// TwinCAT 3 PLC project StageCore
// Title: StageCore
// Company: _
// Author: Krystian Lis et al.
// ProjectVersion: 6.0.0
// ProgramVersion: 3.1.4026.18
// libraries:
//   Tc2_Math, * (Beckhoff Automation GmbH)
//   Tc2_Standard, * (Beckhoff Automation GmbH)
//   Tc2_System, * (Beckhoff Automation GmbH)
//   Tc2_Utilities, * (Beckhoff Automation GmbH)
// project tree:
//   Broadcast/Arg/Args/BOOL/ BoolArg.TcPOU (not stored), IArgToIBoolArg.TcPOU (not stored), I_BoolArg.TcIO (not stored)
//   Broadcast/Arg/Args/DWORD/ DwordArg.TcPOU (not stored), IArgToIDwordArg.TcPOU (not stored), I_DwordArg.TcIO (not stored)
//   Broadcast/Arg/Args/REAL/ IArgToIRealtArg.TcPOU (not stored), I_RealArg.TcIO (not stored), RealArg.TcPOU (not stored)
//   Broadcast/Arg/ IArgToIComp.TcPOU, ICompToIArg.TcPOU (not stored), I_Arg.TcIO (not stored)
//   Broadcast/Callable/ I_Callable.TcIO (not stored)
//   Broadcast/Helpers/ GetSignal.TcPOU (not stored), GetReceiver.TcPOU
//   Broadcast/Receiver/ ICompToIRec.TcPOU (not stored), I_Receiver.TcIO, I_ReceiverNode.TcIO (not stored), Receiver.TcPOU
//   Broadcast/Signal/ ICompToISignal.TcPOU, I_SignalEmit.TcIO, I_Signal.TcIO, I_SignalNode.TcIO (not stored), Signal.TcPOU
//   Broadcast/Sys/Helpers/ _BroadcastDefragment.TcPOU, _BroadcastGetBestFit.TcPOU (not stored), _Emit.TcPOU (not stored), _Pair.TcPOU, _RegSignal.TcPOU (not stored), _Unpair.TcPOU (not stored)
//   Broadcast/Sys/Structs/ _BroadcastStruct.TcDUT (not stored), _BroadcastUnion.TcDUT (not stored)
//   Broadcast/Sys/ _Broadcast.TcGVL (not stored)
//   Dbg/ DebugInfo.TcPOU, NewDebug.TcPOU, DebugMode.TcDUT, I_Debug.TcIO (not stored), _DebugInfo.TcDUT, _Debug.TcGVL
//   Entity/Core/ Component.TcPOU, I_Component.TcIO (not stored), GetOwnerFromRaw.TcPOU, I_RawComponent.TcIO (not stored), I_Entity.TcIO, GetNextEntity.TcPOU, GetPrevEntity.TcPOU
//   Entity/Core/Scope/ EntityEnd.TcPOU, EntityExtend.TcPOU, EntityStart.TcPOU
//   Entity/Sys/ _EntityState.TcDUT (not stored), _Ec.TcGVL
//   Entity/Sys/_Helpers/ _EntityEnd.TcPOU, _EntityExtend.TcPOU (not stored), _EntityStart.TcPOU (not stored), _RegisterComponent.TcPOU
//   Entity/Sys/_Itf/ I_ComponentNode.TcIO, I_EntityNode.TcIO
//   Result/Error/ Err.TcGVL (not stored), GenericResult.TcGVL (not stored)
//   Result/ IsErr.TcPOU (not stored), IsNone.TcPOU (not stored), IsOk.TcPOU, IsFail.TcPOU, IsSome.TcPOU (not stored), IsEnd.TcPOU, Result.TcDUT (not stored), ResultToStr.TcPOU
//   Runtime/Execute/ Execute.TcPOU, I_Execute.TcIO, I_ExecuteNode.TcIO (not stored)
//   Runtime/Init/ Init.TcPOU, I_InitNode.TcIO (not stored), I_Init.TcIO (not stored)
//   Runtime/ Runtime.TcPOU, _Runtime.TcGVL (not stored)
//   State/_Buffer/ _StateBuffer.TcPOU
//   State/Helpers/ GetStateManager.TcPOU, GetState.TcPOU (not stored)
//   State/_Machine/ _StateMachine.TcPOU
//   State/Manager/ ICompToIStateMgr.TcPOU, I_StateManager.TcIO (not stored), StateManager.TcPOU
//   State/State/ ICompToIState.TcPOU (not stored), I_State.TcIO, I_StateInternal.TcIO, State.TcPOU
//   Strings/Alias/ Ch.TcDUT (not stored), Str.TcDUT (not stored)
//   Strings/Strb/ I_Strb.TcIO (not stored), Strb.TcPOU
//   Strings/Strf/ Strf.TcPOU
//   Tags/Casts/ IArgToITag.TcPOU, ICompToITag.TcPOU (not stored)
//   Tags/Helpers/ GetTag.TcPOU, GetTagOption.TcPOU, HasTagOption.TcPOU, HasTag.TcPOU (not stored), MatchPath.TcPOU
//   Tags/ I_Tag.TcIO, I_TagCmp.TcIO, TagBase.TcPOU, TagCmp.TcPOU (not stored), TagPath.TcPOU (not stored), Tag.TcPOU (not stored)
//   Jobs/Worker/Base/ Worker.TcPOU, I_Worker.TcIO
//   Jobs/Worker/ LoopWorker.TcPOU, BlockingWorker.TcPOU
//   Jobs/Job/ I_Job.TcIO, I_JobInternal.TcIO, Job.TcPOU
//   Jobs/ JobState.TcDUT
//   _/ Param.TcGVL
// (motion and I/O tree: see PLC project stageutils)
// real-time tasks:
//   TASK Example: cycle T#10ms, priority 20, ADS port 350
//   TASK Test: cycle T#10ms, priority 21, ADS port 351
//   TASK VISU_TASK: cycle T#200000us, priority 30, ADS port 352

// ---- Dbg/DebugMode.TcDUT
{attribute 'qualified_only'}
{attribute 'strict'}
{attribute 'to_string'}
TYPE DebugMode :
(
	Notify,
	Panic
) BYTE;
END_TYPE

// ---- Dbg/_DebugInfo.TcDUT
TYPE INTERNAL _DebugInfo :
STRUCT
	iDebugMain: I_Debug;
	iDebugSub: I_Debug;
	mode: DebugMode;
	sComment: Str;
END_STRUCT
END_TYPE

// ---- Jobs/JobState.TcDUT
(*
State of a Job.
*)
{attribute 'qualified_only'}
{attribute 'strict'}
TYPE JobState :
(
	Error,
	Idle,
	Enqueue,
	Ready,
	Running,
	Aborted,
	Completed
) BYTE := Idle;
END_TYPE

// ---- Dbg/_Debug.TcGVL
{attribute 'qualified_only'}
VAR_GLOBAL INTERNAL
	debugMsg: ARRAY[1..Param.DEBUG_CAP] OF _DebugInfo;	
	nLastIdx: UDINT;
	
	nTotalNumber: UDINT;
	nNotifyNumber: UDINT;
	nPanicNumber: UDINT;
END_VAR

// ---- Entity/Sys/_Ec.TcGVL
// ---------------------------------------------------------------------------
// GLOBAL DATA BLOCK: _Ec
// Purpose: Stores and manages the state and structure of all registered entities 
//          and tracks the current scope under construction.

// This attribute ensures variables are accessed using qualified names (e.g., _Ec.iFirst)
{attribute 'qualified_only'}

VAR_GLOBAL INTERNAL    
    // Reference to the first registered entity in the global entity list
    iFirst: I_Entity;

    // Reference to the last registered entity in the global entity list
    iLast: I_Entity;

    // Points to the entity currently being constructed
    // Used to add components or nested entities during initialization
    iUnderConstruction: I_Entity;

    // Tracks how many nested entity scopes are currently under construction
    // Used to manage hierarchical or recursive construction logic
    nConstructedScopes: UDINT;
END_VAR

// ---- _/Param.TcGVL
{attribute 'qualified_only'}
// DO NOT SET ANY OF THE CAP PARAMETERS TO 0 OR LARGER THAN MAX DINT!!!
VAR_GLOBAL CONSTANT
	SIGNAL_CAP		: UDINT(1..16#7FFFFFFF) := 20; // Max number of signals.
	RECEIVER_CAP	: UDINT(1..16#7FFFFFFF) := 100; // Max number of signal-receiver pairings.
	
	
	DEBUG_CAP	: UDINT(1..16#7FFFFFFF) := 10; // Max number of debug messages.
	INIT_INTERNAL_DEBUG_MODE: DebugMode := DebugMode.Panic; // Should internal debug messages during initialization stop Runtime?
	EXE_INTERNAL_DEBUG_MODE: DebugMode := DebugMode.Notify; // Should internal debug messages during execution stop Runtime?
END_VAR

// ---- Broadcast/Receiver/I_Receiver.TcIO
(*
Represents a receiver in the Broadcast system. Implements the necessary methods for receiving events and pairing signals.
Can be casted to `I_Component`.
*)
INTERFACE I_Receiver EXTENDS I_ReceiverNode, I_RawComponent

PROPERTY Tag : I_Tag
GET
END_GET
END_PROPERTY

END_INTERFACE

// ---- Broadcast/Signal/I_SignalEmit.TcIO
(*
Enables pairing with receivers and emitting, but not casting to `I_Component`.
*)
INTERFACE I_SignalEmit

(*
Emits an argument through the signal's broadcasting system.  
If no argument is provided, it defaults to emitting the associated tag.
Returns:
- `Ok` - On Success
- `Err.InfLoop` - Upon recursive call attempt
*)
METHOD Emit : Result
VAR_INPUT
	iArg			: I_Arg := 0;
END_VAR
END_METHOD

(*
Emits an argument to a specified receiver.
Returns:
- `Ok` - If the emission is successful.
- `Err.Itf0` - If the receiver interface is invalid.
- `Err.InfLoop` - Upon recursive call attempt
*)
METHOD EmitTo : Result
VAR_INPUT
	iReceiver		: I_Receiver;
	iArg			: I_Arg := 0;
END_VAR
END_METHOD

(*
Allows access to Option property of the internal Tag.
*)
PROPERTY Option : Str
GET
END_GET
SET
END_SET
END_PROPERTY

(*
Pairs the signal with a receiver.  
Returns:
- `Ok` - If pairing is successful.
- `Err.Itf0` - If the receiver interface is invalid.
- `Err.IncArg` - If the `I_Receiver` is invalid.
- `Err.ItfEq` - If the `I_Receiver` is already paired with this `I_Signal`.
- `Err.Ovf` - If there is no space for another pairing.
*)
METHOD Pair : Result
VAR_INPUT
	iReceiver		: I_Receiver;
END_VAR
END_METHOD

(*
Provides access to the tag associated with the signal.
*)
PROPERTY Tag : I_Tag
GET
END_GET
END_PROPERTY

(*
Unpairs the signal from a specified receiver.
Returns:
- `Ok` - If unpairing is successful.
- `Err.Itf0` - If the receiver interface is invalid.
- `Err.IncArg` - If the `I_Receiver` is invalid.
- `Err.NoMatch` - If `I_Signal` is not paired with this `I_Receiver`.
*)
METHOD Unpair : Result
VAR_INPUT
	iReceiver		: I_Receiver;
END_VAR
END_METHOD

END_INTERFACE

// ---- Broadcast/Signal/I_Signal.TcIO
(*
Enables pairing with receivers and casting to `I_Component`, but no emitting.
*)
INTERFACE I_Signal EXTENDS I_Debug, I_RawComponent

(*
Pairs the signal with a receiver.  
Returns:
- `Ok` - If pairing is successful.
- `Err.Itf0` - If the receiver interface is invalid.
- `Err.IncArg` - If the `I_Receiver` is invalid.
- `Err.ItfEq` - If the `I_Receiver` is already paired with this `I_Signal`.
- `Err.Ovf` - If there is no space for another pairing.
*)
METHOD Pair : Result
VAR_INPUT
	iReceiver		: I_Receiver;
END_VAR
END_METHOD

PROPERTY Tag : I_Tag
GET
END_GET
END_PROPERTY

(*
Unpairs the signal from a specified receiver.
Returns:
- `Ok` - If unpairing is successful.
- `Err.Itf0` - If the receiver interface is invalid.
- `Err.IncArg` - If the `I_Receiver` is invalid.
- `Err.NoMatch` - If `I_Signal` is not paired with this `I_Receiver`.
*)
METHOD Unpair : Result
VAR_INPUT
	iReceiver		: I_Receiver;
END_VAR
END_METHOD

END_INTERFACE

// ---- Entity/Core/I_Entity.TcIO
(*
Represents a registered entity in the Entity-Component system.
*)
INTERFACE I_Entity EXTENDS I_EntityNode

END_INTERFACE

// ---- Entity/Sys/_Itf/I_ComponentNode.TcIO
INTERFACE INTERNAL I_ComponentNode EXTENDS I_Debug

PROPERTY INTERNAL _Entity : I_Entity
GET
END_GET
SET
END_SET
END_PROPERTY

PROPERTY INTERNAL _Next : I_Component
GET
END_GET
SET
END_SET
END_PROPERTY

PROPERTY INTERNAL _Prev : I_Component
GET
END_GET
SET
END_SET
END_PROPERTY

END_INTERFACE

// ---- Entity/Sys/_Itf/I_EntityNode.TcIO
INTERFACE INTERNAL I_EntityNode EXTENDS I_Debug

PROPERTY INTERNAL _FirstComp : I_Component
GET
END_GET
SET
END_SET
END_PROPERTY

PROPERTY INTERNAL _LastComp : I_Component
GET
END_GET
SET
END_SET
END_PROPERTY

PROPERTY INTERNAL _Next : I_Entity
GET
END_GET
SET
END_SET
END_PROPERTY

PROPERTY INTERNAL _Prev : I_Entity
GET
END_GET
SET
END_SET
END_PROPERTY

PROPERTY INTERNAL _Size : UDINT
GET
END_GET
SET
END_SET
END_PROPERTY

PROPERTY INTERNAL _State : _EntityState
GET
END_GET
SET
END_SET
END_PROPERTY

(*
Description: Retrieves a previous component before the inputted one or last component if referenced value is 0.
Returns:
- Ok - Returns upon success, updates referenced value with new component.
- Err.InvRef - Invalid output reference.
- Err.ItfEq - Provided interface pointer doesn't belong to the queried entity. Nulls reference.
- Err.NotFound - The entity doesn't contain any components. Nulls reference.
- Err.End - No more components. Nulls reference.
*)
METHOD GetNextComp : Result
VAR_INPUT
	iOut		: REFERENCE TO I_Component;
END_VAR
END_METHOD

(*
Description: Retrieves a previous component before the inputted one or last component if referenced value is 0.
Returns:
- Ok - Returns upon success, updates referenced value with new component.
- Err.InvRef - Invalid output reference.
- Err.ItfEq - Provided interface pointer doesn't belong to the queried entity. Nulls reference.
- Err.NotFound - The entity doesn't contain any components. Nulls reference.
- Err.End - No more components. Nulls reference.
*)
METHOD GetPrevComp : Result
VAR_INPUT
	iOut		: REFERENCE TO I_Component;
END_VAR
END_METHOD

(*
Provides the size of the entity, indicating the number of components it manages.  
Note: For internal logic purposes, this value is incremented by one beyond the actual component count.
*)
PROPERTY Size : UDINT
GET
END_GET
END_PROPERTY

END_INTERFACE

// ---- Runtime/Execute/I_Execute.TcIO
(*
A `Execute` method of FB implmenting this interface will be called every control loop cycle.
*)
INTERFACE I_Execute EXTENDS I_Debug

(*
If registered, this method will be executed cyclically.
*)
METHOD Execute
VAR_INPUT
	nPhase: INT;
END_VAR
END_METHOD

END_INTERFACE

// ---- State/State/I_State.TcIO
(*
Allows states to be cast to `I_RawComponent`.
*)
INTERFACE I_State EXTENDS I_RawComponent, I_Debug, I_StateInternal

(*
Returns the entity that owns this state.
*)
PROPERTY Owner : I_Entity
GET
END_GET
END_PROPERTY

PROPERTY Tag : I_Tag
GET
END_GET
END_PROPERTY

END_INTERFACE

// ---- State/State/I_StateInternal.TcIO
INTERFACE INTERNAL I_StateInternal

METHOD INTERNAL _CanActivate : BOOL
VAR_INPUT
END_VAR
END_METHOD

METHOD INTERNAL _CanDeactivate : BOOL
VAR_INPUT
END_VAR
END_METHOD

PROPERTY INTERNAL _InQueue : BOOL
GET
END_GET
SET
END_SET
END_PROPERTY

PROPERTY INTERNAL _NextInBuffer : I_State
GET
END_GET
SET
END_SET
END_PROPERTY

METHOD INTERNAL _OnEntry
VAR_INPUT
END_VAR
END_METHOD

METHOD INTERNAL _OnExecute
VAR_INPUT
END_VAR
END_METHOD

METHOD INTERNAL _OnExit
VAR_INPUT
END_VAR
END_METHOD

(*
Returns the entity that owns this state.
*)
PROPERTY Owner : I_Entity
GET
END_GET
END_PROPERTY

END_INTERFACE

// ---- Tags/I_Tag.TcIO
(*
An identifier that uses reflection to generate a unique symbol path.
It simplifies the path by removing project, PLC, and tag segments.
Can be casted to `I_Arg` and `I_Component`.
Example:
- Reflection: proj.plc.MAIN.functionBlock[*]._tag
- Path: MAIN.functionBlock.5
*)
INTERFACE I_Tag EXTENDS I_Debug, I_RawComponent, I_Arg

// Read address path without Option segment.
PROPERTY Id : Str
GET
END_GET
END_PROPERTY

// Modify or read the optional segment.
PROPERTY Option : Str
GET
END_GET
END_PROPERTY

END_INTERFACE

// ---- Tags/I_TagCmp.TcIO
(*
A tool for performing CASE OF-like evaluations on `I_Tag`.  
It enables sequential evaluation of conditions and stops when `IsTrue`, `IsFalse`, or `IsErr` methods are invoked.
Allows method chaining.
*)
INTERFACE INTERNAL I_TagCmp

(*
Updates its internal state based on the internal status and option.  
Sets the state to `Ok` if the base tag is `Ok` and has the specified Option; otherwise, sets the state to `None`.
*)
METHOD AndHasOption : I_TagCmp
VAR_INPUT
	sOption		: Str;
END_VAR
END_METHOD

(*
Updates its internal state based on the internal status and an external condition.  
Sets the state to `Ok` if the base tag is `Ok` and the external condition is TRUE; otherwise, sets the state to `None`.
*)
METHOD AndIf : I_TagCmp
VAR_INPUT
	bCondition: BOOL;
END_VAR
END_METHOD

(*
Updates its internal state based on the internal status and option.  
Sets the state to `Ok` if the base tag has the specified Option.
*)
METHOD HasOption : I_TagCmp
VAR_INPUT
	sOption		: Str;
END_VAR
END_METHOD

(*
Returns `TRUE` if any evaluated conditions resulted in `Error`.  
Halts further evaluations by locking the current state.
*)
METHOD IsErr : BOOL
VAR_INPUT
END_VAR
END_METHOD

(*
Returns `TRUE` if all evaluated conditions resulted in `FALSE`.  
Halts further evaluations by locking the current state.
*)
METHOD IsFalse : BOOL
VAR_INPUT
END_VAR
END_METHOD

(*
Returns `TRUE` if any evaluated condition resulted in `TRUE`.  
Halts further evaluations by locking the current state.
*)
METHOD IsTrue : BOOL
VAR_INPUT
END_VAR
END_METHOD

(*
Updates its internal state based on the internal status and external I_Tag.  
Sets the state to `Ok` if the base tag matches the external tag.
*)
METHOD Match : I_TagCmp
VAR_INPUT
	iOther: I_Tag;
END_VAR
END_METHOD

(*
Updates its internal state based on the internal status and a string value.  
Sets the state to `Ok` if the base tag Id matches the provided string from right to left.
*)
METHOD MatchId : I_TagCmp
VAR_INPUT
	sIdToMatch		: Str;
END_VAR
END_METHOD

(*
Updates its internal state based on the internal status and a string value.  
Sets the state to `Ok` if the base tag Id matches the provided string pattern.
Allows wildcards.
*)
METHOD MatchWcdId : I_TagCmp
VAR_INPUT
	sPattern 			: Str;
END_VAR
END_METHOD

(*
Updates its internal state based on the internal status and an external condition.  
Sets the state to `Ok` if the base tag is `Ok` or the external condition is TRUE.
*)
METHOD OrIf : I_TagCmp
VAR_INPUT
	bCondition: BOOL;
END_VAR
END_METHOD

(*
Sets a new base tag for comparison and resets the result and lock states.
Fails if `iBaseTag` is `0`;
*)
METHOD Set : I_TagCmp
VAR_INPUT
	iBaseTag	: I_Tag;
END_VAR
END_METHOD

(*
Updates its internal state based on the internal status and an external condition.  
Sets the state to `Ok` if the base tag is `Ok` xor the external condition is TRUE.
*)
METHOD XorIf : I_TagCmp
VAR_INPUT
	bCondition: BOOL;
END_VAR
END_METHOD

END_INTERFACE

// ---- Jobs/Worker/Base/I_Worker.TcIO
(*
An interface that represents an object that schedules jobs execution.
*)
INTERFACE I_Worker EXTENDS I_Debug

(*
Defer the Job. Move it to the end of queue.
Returns:
- Ok - Success
- Err.Itf0 - iJob = 0
- Err.NoMatch = iJob.Worker <> THIS^
*)
METHOD Defer : Result
VAR_INPUT
    iJob : I_Job;
END_VAR
END_METHOD

(*
Remove job from the queue and resets it.
Returns:
- Ok - Success
- Err.Itf0 - iJob = 0
- Err.NoMatch - iJob.Worker <> THIS^
- Err.IncArg - iJob.State = TaskState.Idle
*)
METHOD Dequeue : Result
VAR_INPUT
	iJob: I_Job;
END_VAR
END_METHOD

(*
Add Job to queue.
Returns:
- Ok - Success
- Err.Itf0 - iJob = 0
- Err.NoMatch - iJob.Worker <> THIS^
- Err.IncArg - iJob.State <> TaskState.Idle 
*)
METHOD Enqueue : Result
VAR_INPUT
	iJob: I_Job;
END_VAR
END_METHOD

(*
Returns first the Job in queue.
*)
PROPERTY First : I_Job
GET
END_GET
END_PROPERTY

END_INTERFACE

// ---- Jobs/Job/I_Job.TcIO
(*
Allow others to start and abort job.
*)
INTERFACE I_Job EXTENDS I_JobInternal

(*
Notifies scheduler to aboort this job.
Returns Err.IncArg on State = Idle
*)
METHOD Abort : Result
VAR_INPUT
END_VAR
END_METHOD

(*
Starts the job and adds it to Workers queue.
Returns Err.IncArg on State <> Idle.
Returns Err.Itf0 on Worker = 0.
*)
METHOD Start : Result
VAR_INPUT
END_VAR
END_METHOD

END_INTERFACE

// ---- Jobs/Job/I_JobInternal.TcIO
INTERFACE INTERNAL I_JobInternal EXTENDS I_Debug

PROPERTY INTERNAL _Next : I_Job
GET
END_GET
SET
END_SET
END_PROPERTY

METHOD INTERNAL _OnAbort
VAR_INPUT
END_VAR
END_METHOD

METHOD INTERNAL _OnDone
VAR_INPUT
END_VAR
END_METHOD

METHOD INTERNAL _OnExit
VAR_INPUT
END_VAR
END_METHOD

METHOD INTERNAL _OnRun
VAR_INPUT
END_VAR
END_METHOD

METHOD INTERNAL _OnStart
VAR_INPUT
END_VAR
END_METHOD

PROPERTY INTERNAL _Prev : I_Job
GET
END_GET
SET
END_SET
END_PROPERTY

(*
Returns Jobs state
*)
PROPERTY State : JobState
GET
END_GET
END_PROPERTY

(*
Returns Worker working on this job
*)
PROPERTY Worker : I_Worker
GET
END_GET
END_PROPERTY

END_INTERFACE

// ---- State/State/State.TcPOU
(*
An abstract representation of a system state, providing the foundation for implementing state-specific behavior.  
Manages its owner entity and supports state transitions within the system.  
Offers default behavior for state lifecycle methods, allowing programmers to override only the relevant parts.
*)
FUNCTION_BLOCK ABSTRACT State IMPLEMENTS I_StateInternal, I_State
VAR
	{attribute 'hide'}
	_comp						: Component(THIS^);
	{attribute 'hide'}
	_bInQueue					: BOOL;
	{attribute 'hide'}
	_iNextInBuffer				: I_State; // State Buffer management
	
	_tag			: TagBase;	
END_VAR

METHOD INTERNAL _CanActivate : BOOL
_CanActivate := CanActivate();
END_METHOD

METHOD INTERNAL _CanDeactivate : BOOL
_CanDeactivate := CanDeactivate();
END_METHOD

PROPERTY INTERNAL _InQueue : BOOL
GET
_InQueue := _bInQueue;
END_GET
SET
_bInQueue := _InQueue;
END_SET
END_PROPERTY

PROPERTY INTERNAL _NextInBuffer : I_State
GET
_NextInBuffer := _iNextInBuffer;
END_GET
SET
_iNextInBuffer := _NextInBuffer;
END_SET
END_PROPERTY

METHOD INTERNAL _OnEntry
OnEntry();
END_METHOD

METHOD INTERNAL _OnExecute
OnExecute();
END_METHOD

METHOD INTERNAL _OnExit
OnExit();
END_METHOD

(*
Determines whether the state can be activated.  
Returns `TRUE` by default but can be overridden for specific activation conditions.
*)
METHOD PROTECTED CanActivate : BOOL
VAR_INPUT
END_VAR
CanActivate := TRUE;
END_METHOD

(*
Determines whether the state can be deactivated.  
Returns `TRUE` by default but can be overridden for specific deactivation conditions.
*)
METHOD PROTECTED CanDeactivate : BOOL
VAR_INPUT
END_VAR
CanDeactivate := TRUE;
END_METHOD

//FB_Init is always available implicitly and it is used primarily for initialization.
//The return value is not evaluated. For a specific influence, you can also declare the
//methods explicitly and provide additional code there with the standard initialization
//code. You can evaluate the return value.
{attribute 'hide'}
METHOD FB_Init: BOOL
VAR_INPUT
    bInitRetains: BOOL; // TRUE: the retain variables are initialized (reset warm / reset cold)
    bInCopyCode: BOOL;  // TRUE: the instance will be copied to the copy code afterward (online change)   
END_VAR
END_METHOD

(*
Executed when the state is entered.  
Provides a hook for defining state-specific behavior to be performed during the transition into this state.
*)
METHOD PROTECTED OnEntry
VAR_INPUT
END_VAR
END_METHOD

(*
Executed during the state's operation.  
Used to define state-specific logic that runs while the state is active.
*)
METHOD PROTECTED OnExecute
VAR_INPUT
END_VAR
END_METHOD

(*
Executed when the state transitions to another state.  
Provides a hook for defining cleanup or transition-specific behavior.
*)
METHOD PROTECTED OnExit
VAR_INPUT
END_VAR
END_METHOD

(*
Returns the entity that owns this state.
*)
PROPERTY FINAL Owner : I_Entity
GET
Owner := _comp.Entity;
END_GET
END_PROPERTY

(*
Allows initializing an external interface variable with an interface pointer to this instance within declaration block.
Example:
iState: I_State;
state: SomeState := (Proxy := iState);
Result: iState <> 0 
*)
PROPERTY Proxy : REFERENCE TO I_State
SET
Proxy := THIS^;
END_SET
END_PROPERTY

(*
Provides access to the `I_Tag` associated with the state.
*)
PROPERTY FINAL Tag : I_Tag
GET
Tag := _tag;
END_GET
END_PROPERTY

END_FUNCTION_BLOCK

// ---- Entity/Core/Component.TcPOU
(*
Allows registration of FB implementing I_RawComponent. The framework will automatically add this function block to the entity's scope. Implements I_Component.
*)
FUNCTION_BLOCK FINAL Component IMPLEMENTS I_Component
VAR
	_iComponent: I_RawComponent;
	_iEntity: I_Entity;
	_iNext: I_Component;
	_iPrev: I_Component;			
END_VAR

PROPERTY _Entity : I_Entity
GET
_Entity := _iEntity;
END_GET
SET
_iEntity := _Entity;
END_SET
END_PROPERTY

PROPERTY _Next : I_Component
GET
_Next := _iNext;
END_GET
SET
_iNext := _Next;
END_SET
END_PROPERTY

PROPERTY _Prev : I_Component
GET
_Prev := _iPrev;
END_GET
SET
_iPrev := _Prev;
END_SET
END_PROPERTY

(*
Returns parent Entity.
*)
PROPERTY Entity : I_Entity
GET
Entity := _iEntity;
END_GET
END_PROPERTY

//FB_Init is always available implicitly and it is used primarily for initialization.
//The return value is not evaluated. For a specific influence, you can also declare the
//methods explicitly and provide additional code there with the standard initialization
//code. You can evaluate the return value.
{attribute 'hide'}
METHOD FB_init: BOOL
VAR_INPUT
    bInitRetains: BOOL; // TRUE: the retain variables are initialized (reset warm / reset cold)
    bInCopyCode: BOOL;  // TRUE: the instance will be copied to the copy code afterward (online change)
	
	iComponent		: I_RawComponent;
END_VAR
VAR
	_nResult		: Result;
END_VAR
_iComponent := iComponent;

IF _Ec.iUnderConstruction = 0 THEN
	NewDebug(THIS^, Param.INIT_INTERNAL_DEBUG_MODE, 'Declared outside Entity scope!');
	RETURN;
END_IF
			
IF IsErr(_RegisterComponent(THIS^), nOut => _nResult) THEN
	NewDebug(THIS^, Param.INIT_INTERNAL_DEBUG_MODE, Tc2_Standard.CONCAT('Failed with code: ', ResultToStr(_nResult)));
END_IF
END_METHOD

(*
Returns raw I_RawComponent pointer.
*)
PROPERTY Raw : I_RawComponent
GET
Raw := _iComponent;
END_GET
END_PROPERTY

END_FUNCTION_BLOCK

// ---- Dbg/NewDebug.TcPOU
(*
Logs a debug message as a string tied to a `I_Debug` interface for inspection and troubleshooting within the IDE.
*)
FUNCTION NewDebug
VAR_INPUT
	iDebugMain: I_Debug;
	mode: DebugMode;
	sComment: Str;
	iDebugSub: I_Debug := 0;
END_VAR

IF _Debug.nLastIdx < Param.DEBUG_CAP THEN
	_Debug.nLastIdx := _Debug.nLastIdx + 1;
ELSE
	_Debug.nLastIdx := 1;
END_IF

_Debug.nTotalNumber := _Debug.nTotalNumber + 1;

CASE mode OF
	DebugMode.Notify:
		_Debug.nNotifyNumber := _Debug.nNotifyNumber + 1;
	DebugMode.Panic:	
		_Debug.nPanicNumber := _Debug.nPanicNumber + 1;
END_CASE

_Debug.debugMsg[_Debug.nLastIdx].iDebugMain := iDebugMain;
_Debug.debugMsg[_Debug.nLastIdx].iDebugSub := iDebugSub;
_Debug.debugMsg[_Debug.nLastIdx].sComment := sComment;
_Debug.debugMsg[_Debug.nLastIdx].mode := mode;

END_FUNCTION

// ---- Entity/Sys/_Helpers/_RegisterComponent.TcPOU
FUNCTION INTERNAL _RegisterComponent : Result
VAR_INPUT
    iComponent  : I_Component;
END_VAR

// Check if the runtime system has been initialized
IF NOT _Runtime.bInit THEN
    // If not initialized, return with an initialization error
    _RegisterComponent := Err.Init;
    RETURN;
END_IF

// Validate that there is an entity currently under construction and the component reference is valid
IF _Ec.iUnderConstruction = 0 OR iComponent = 0 THEN
    // If either is invalid, return interface error
    _RegisterComponent := Err.Itf0;
    RETURN;
END_IF

// Ensure the entity under construction is in the 'Registered' state
IF _Ec.iUnderConstruction._State <> _EntityState.Registered THEN
    // If not registered, the entity context is invalid for component registration
    _RegisterComponent := Err.NotFound;
    RETURN;
END_IF

// Ensure the component is not already assigned to another entity
IF iComponent._Entity <> 0 THEN
    // Component is already linked to an entity, return incorrect argument error
    _RegisterComponent := Err.IncArg;
    RETURN;
END_IF

// Add entity as parent
iComponent._Entity := _Ec.iUnderConstruction;
iComponent._Entity._Size := iComponent._Entity._Size + 1;

// If the entity already has components, append this one to the end of the component list
IF _Ec.iUnderConstruction._LastComp <> 0 THEN
    _Ec.iUnderConstruction._LastComp._Next := iComponent;           // Link previous last to new component
    iComponent._Prev := _Ec.iUnderConstruction._LastComp;           // Link new component back to previous last
    _Ec.iUnderConstruction._LastComp := iComponent;                 // Update the last component pointer
    _RegisterComponent := Ok;

// If this is the first component being added, initialize the list
ELSE
    _Ec.iUnderConstruction._FirstComp := iComponent;                // Set as first component
    _Ec.iUnderConstruction._LastComp := iComponent;                 // Also set as last component
    _RegisterComponent := Ok;
END_IF

END_FUNCTION

// ---- Runtime/Init/Init.TcPOU
(*
Allows registration of FB implementing `I_Init`. 
*)
FUNCTION_BLOCK FINAL Init IMPLEMENTS I_InitNode, I_Debug
VAR
	_iInit			: I_Init;
	_iNext			: I_InitNode;
	_nState			: Result;
	_nPhase			: INT;
END_VAR

METHOD INTERNAL Attach : Result
VAR_INPUT
	iInit			: I_InitNode;
END_VAR
VAR
	_iThis			: I_InitNode := THIS^;
END_VAR
IF iInit = 0 THEN
	NewDebug(THIS^, Param.INIT_INTERNAL_DEBUG_MODE, Tc2_Standard.CONCAT(__POUNAME(), ': Itf = 0!'));
	RETURN;
END_IF

IF _iThis <> _Runtime.iLastInit THEN
	NewDebug(THIS^, Param.INIT_INTERNAL_DEBUG_MODE, Tc2_Standard.CONCAT(__POUNAME(), ': Is not the last node!'));
	RETURN;
END_IF

IF IsSome(iInit.state) THEN
	NewDebug(iInit, Param.INIT_INTERNAL_DEBUG_MODE, Tc2_Standard.CONCAT(__POUNAME(), ': Has already been added!'));
	RETURN;
END_IF

_Runtime.iLastInit := iInit;
_iNext := iInit;
END_METHOD

//FB_Init is always available implicitly and it is used primarily for initialization.
//The return value is not evaluated. For a specific influence, you can also declare the
//methods explicitly and provide additional code there with the standard initialization
//code. You can evaluate the return value.
{attribute 'hide'}
METHOD FB_Init: BOOL
VAR_INPUT
    bInitRetains: BOOL; // TRUE: the retain variables are initialized (reset warm / reset cold)
    bInCopyCode: BOOL;  // TRUE: the instance will be copied to the copy code afterward (online change)
	
	iInit			: I_Init;
END_VAR
IF IsSome(_nState) THEN
	RETURN;
END_IF

IF (_iInit := iInit) = 0 THEN
	_nState := Err.Itf0;
	NewDebug(THIS^, Param.INIT_INTERNAL_DEBUG_MODE, Tc2_Standard.CONCAT(__POUNAME(), ': Itf = 0!'));
	RETURN;
END_IF



IF _Runtime.iLastInit <> 0 THEN
	IF IsErr(_Runtime.iLastInit.Attach(THIS^), nOut => _nState) THEN
		NewDebug(THIS^, Param.INIT_INTERNAL_DEBUG_MODE, Tc2_Standard.CONCAT(__POUNAME(), ': Error inside!'));
	END_IF
ELSE
	_Runtime.iFirstInit := THIS^;
	_Runtime.iLastInit := THIS^;
	_nState := Ok;
END_IF
END_METHOD

METHOD INTERNAL Init
VAR_OUTPUT
	iNext: I_InitNode;
END_VAR
_iInit.Init(_nPhase);
iNext := _iNext;
END_METHOD

PROPERTY Phase : INT
GET
Phase := _nPhase;
END_GET
SET
_nPhase := Phase;
END_SET
END_PROPERTY

PROPERTY INTERNAL State : Result
GET
State := _nState;
END_GET
SET
IF IsNone(_nState) THEN
	_nState := State;
END_IF
END_SET
END_PROPERTY

END_FUNCTION_BLOCK

// ---- Result/ResultToStr.TcPOU
// Converts a Result value to its corresponding string representation.
// Returns a string that describes the given Result value.
FUNCTION ResultToStr : Str
VAR_INPUT
    nResult : Result; // Result variable to convert to a string
END_VAR

CASE nResult OF
    Ok: ResultToStr := 'Ok';
    None: ResultToStr := 'None';
    Error: ResultToStr := 'Error';
    Err.Itf0: ResultToStr := 'Itf0';
    Err.Str0: ResultToStr := 'Str0';
    Err.ItfEq: ResultToStr := 'ItfEq';
    Err.NoMatch: ResultToStr := 'NoMatch';
    Err.Ptr0: ResultToStr := 'Ptr0';
    Err.InvRef: ResultToStr := 'InvRef';
    Err.Ovf: ResultToStr := 'Ovf';
    Err.Udf: ResultToStr := 'Udf';
    Err.Idx: ResultToStr := 'Idx';
    Err.TcLib: ResultToStr := 'TcLib';
    Err.InfLoop: ResultToStr := 'InfLoop';
    Err.IncArg: ResultToStr := 'IncArg';
	Err.Init: ResultToStr := 'Init';
	Err.NotFound: ResultToStr := 'Item not found';
	Err.InvItf: ResultToStr := 'InvItf';
    Err.End: ResultToStr := 'End';
	ELSE
        ResultToStr := Tc2_Standard.CONCAT('Unknown result: ', INT_TO_STRING(nResult));
END_CASE

END_FUNCTION

// ---- Tags/TagBase.TcPOU
(*
An identifier that uses reflection to generate a unique symbol path.
It simplifies the path by removing project, PLC, and tag segments.
Example:
- Reflection: proj.plc.MAIN.functionBlock[*]._tag
- Path: MAIN.functionBlock.5

TagBase is not component!
*)
{attribute 'reflection'}
FUNCTION_BLOCK TagBase IMPLEMENTS I_Tag
VAR
	{attribute 'instance-path'} 
    {attribute 'noinit'} 
	_sId			: Str;
	_nOptionPos		: USINT;
	_nOptionLen		: USINT;
END_VAR

{attribute 'hide'}
METHOD FB_init : BOOL
VAR_INPUT
	bInitRetains : BOOL; // if TRUE, the retain variables are initialized (warm start / cold start)
	bInCopyCode : BOOL;  // if TRUE, the instance afterwards gets moved into the copy code (online change)
END_VAR
VAR
	i				: INT;
	_sChar			: Ch;
END_VAR
// Delete this name
FOR i := Tc2_Standard.LEN(_sId) TO 1 BY -1 DO
	IF Tc2_Standard.MID(_sId, 1, i) = '.' THEN
		_sId := Tc2_Standard.LEFT(_sId, i - 1);
		EXIT;
	END_IF
END_FOR

// Delete project name
FOR i := 1 TO Tc2_Standard.LEN(_sId) DO
	IF Tc2_Standard.MID(_sId, 1, i) = '.' THEN
		_sId := Tc2_Standard.DELETE(_sId, i, 1);
		EXIT;
	END_IF
END_FOR

// Delete plc name
FOR i := 1 TO Tc2_Standard.LEN(_sId) DO
	IF Tc2_Standard.MID(_sId, 1, i) = '.' THEN
		_sId := Tc2_Standard.DELETE(_sId, i, 1);
		EXIT;
	END_IF
END_FOR

// Replace '[' with '.' and remove ']' 
FOR i := 1 TO Tc2_Standard.LEN(_sId) DO
	_sChar := Tc2_Standard.MID(_sId, 1, i);
	IF _sChar = '[' THEN
		_sId := Tc2_Standard.REPLACE(_sId, '.', 1, i);
	ELSIF _sChar = ']' THEN
		_sId := Tc2_Standard.DELETE(_sId, 1, i);
	END_IF
END_FOR

_sId := Tc2_Utilities.F_ToLCase(_sID);
END_METHOD

// Read address path without Option segment.
PROPERTY Id : Str
GET
IF _nOptionPos <> 0 THEN
	Id := Tc2_Standard.DELETE(_sId, _nOptionLen + 1, _nOptionPos); 
ELSE
	Id := _sId;
END_IF
END_GET
END_PROPERTY

// Modify or read the optional segment.
PROPERTY Option : Str
GET
VAR
	i				: INT;
END_VAR
IF _nOptionPos <> 0 THEN
	Option := Tc2_Standard.DELETE(_sId, _nOptionPos, 1); 
ELSE
	Option := '';
END_IF
END_GET
SET
IF Option <> '' THEN
    _nOptionLen := INT_TO_USINT(Tc2_Standard.LEN(Option));    
    IF _nOptionPos <> 0 THEN
        _sId := Tc2_Standard.LEFT(_sId, _nOptionPos);
        _sId := Tc2_Standard.CONCAT(_sId, Option);
    ELSE
        // The option does not exist, so we append it
        _nOptionPos := INT_TO_USINT(Tc2_Standard.LEN(_sId) + 1);
        _sId := Tc2_Standard.CONCAT(_sId, '.');
        _sId := Tc2_Standard.CONCAT(_sId, Option);
    END_IF
ELSIF _nOptionPos <> 0 THEN
    _sId := Tc2_Standard.LEFT(_sId, _nOptionPos - 1);
    _nOptionPos := 0;
END_IF
END_SET
END_PROPERTY

(*
Allows initializing an external interface variable with an interface pointer to this instance within declaration block.
Example:
iTag: I_Tag;
tag: Tag := (Proxy := iTag);
Result: iTag <> 0 
*)
PROPERTY Proxy : REFERENCE TO I_Tag
SET
Proxy := THIS^;
END_SET
END_PROPERTY

// Return interface pointer to THIS^.
PROPERTY Self : I_Tag
GET
Self := THIS^;
END_GET
END_PROPERTY

END_FUNCTION_BLOCK

// ---- Broadcast/Signal/Signal.TcPOU
(*
Represents a signal node within the Broadcast system.  
Enables the emission of events and supports pairing with receivers.
*)
FUNCTION_BLOCK FINAL Signal IMPLEMENTS I_SignalNode, I_Signal, I_SignalEmit
VAR
	_comp			: Component(THIS^);
	_tag			: TagBase;	
	_nId			: UDINT;
	_nStart			: UDINT;
	_nEnd			: UDINT;
	_nSize			: UDINT;
	_bIsLocked		: BOOL;
END_VAR

PROPERTY INTERNAL _End : UDINT
GET
_End := _nEnd;
END_GET
SET
_nEnd := _End;
END_SET
END_PROPERTY

PROPERTY INTERNAL _Id : UDINT
GET
_Id := _nId;
END_GET
END_PROPERTY

PROPERTY INTERNAL _Size : UDINT
GET
_Size := _nSize;
END_GET
SET
_nSize := _Size;
END_SET
END_PROPERTY

PROPERTY INTERNAL _Start : UDINT
GET
_Start := _nStart;
END_GET
SET
_nStart := _Start;
END_SET
END_PROPERTY

(*
Emits an argument through the signal's broadcasting system.  
If no argument is provided, it defaults to emitting the associated tag.
Returns:
- Ok - On Success
- Err.InfLoop - Upon recursive call attempt
*)
METHOD Emit : Result
VAR_INPUT
	iArg			: I_Arg := 0;
END_VAR
IF _bIsLocked THEN
	Emit := Err.InfLoop;
	RETURN;
END_IF

IF iArg = 0 THEN
	iArg := _tag;
END_IF

_bIsLocked := TRUE;
_Emit(THIS^, iArg);
_bIsLocked := FALSE;

Emit := Ok;
END_METHOD

(*
Emits an argument to a specified receiver.
Returns:
- `Ok` - If the emission is successful.
- `Err.Itf0` - If the receiver interface is invalid.
- `Err.InfLoop` - Upon recursive call attempt
*)
METHOD EmitTo : Result
VAR_INPUT
	iReceiver		: I_Receiver;
	iArg			: I_Arg := 0;
END_VAR
IF iReceiver = 0 THEN
	EmitTo := Err.Itf0;
	RETURN;
END_IF

IF _bIsLocked THEN
	EmitTo := Err.InfLoop;
	RETURN;
END_IF

IF iArg = 0 THEN
	iArg := _tag;
END_IF

_bIsLocked := TRUE;
iReceiver.Receive(iArg);
_bIsLocked := FALSE;

EmitTo := Ok;
END_METHOD

//FB_Init is always available implicitly and it is used primarily for initialization.
//The return value is not evaluated. For a specific influence, you can also declare the
//methods explicitly and provide additional code there with the standard initialization
//code. You can evaluate the return value.
{attribute 'hide'}
METHOD FB_Init: BOOL
VAR_INPUT
    bInitRetains: BOOL; // TRUE: the retain variables are initialized (reset warm / reset cold)
    bInCopyCode: BOOL;  // TRUE: the instance will be copied to the copy code afterward (online change)   
END_VAR
VAR
	_r	: Result;
END_VAR
CASE (_r := _RegSignal(THIS^, nIndex => _nId)) OF
	Ok:
		// Ignore
	Err.Ovf:
		NewDebug(THIS^, Param.INIT_INTERNAL_DEBUG_MODE, '_Broadcast.iSignal table overflow!');
	ELSE
		NewDebug(THIS^, Param.INIT_INTERNAL_DEBUG_MODE, TC2_Standard.CONCAT('_RegSignal(I_Signal): unknown error! Error code: ', TO_STRING(_r)));
END_CASE
END_METHOD

(*
Allows access to Option property of the internal Tag.
*)
PROPERTY Option : Str
GET
Option := _tag.Option;
END_GET
SET
_tag.Option := Option;
END_SET
END_PROPERTY

(*
Pairs the signal with a receiver.  
Returns:
- `Ok` - If pairing is successful.
- `Err.Itf0` - If the receiver interface is invalid.
- `Err.IncArg` - If the `I_Receiver` is invalid.
- `Err.ItfEq` - If the `I_Receiver` is already paired with this `I_Signal`.
- `Err.Ovf` - If there is no space for another pairing.
*)
METHOD Pair : Result
VAR_INPUT
	iReceiver		: I_Receiver;
END_VAR
IF iReceiver = 0 THEN
	Pair := Err.Itf0;
ELSE
	Pair := _Pair(THIS^, iReceiver);
END_IF
END_METHOD

(*
Allows initializing an external interface variable with an interface pointer to this instance within declaration block.
Example:
iSignal: I_Signal;
signal: Signal := (Proxy := iSignal);
Result: iSignal <> 0 
*)
PROPERTY Proxy : REFERENCE TO I_SignalEmit
SET
Proxy := THIS^;
END_SET
END_PROPERTY

(*
Provides access to the tag associated with the signal.
*)
PROPERTY Tag : I_Tag
GET
Tag := _tag;
END_GET
END_PROPERTY

(*
Unpairs the signal from a specified receiver.
Returns:
- `Ok` - If unpairing is successful.
- `Err.Itf0` - If the receiver interface is invalid.
- `Err.IncArg` - If the `I_Receiver` is invalid.
- `Err.NoMatch` - If `I_Signal` is not paired with this `I_Receiver`.
*)
METHOD Unpair : Result
VAR_INPUT
	iReceiver		: I_Receiver;
END_VAR
IF iReceiver = 0 THEN
	Unpair := Err.Itf0;
ELSE
	Unpair := _Unpair(THIS^, iReceiver);
END_IF
END_METHOD

END_FUNCTION_BLOCK

// ---- Broadcast/Sys/Helpers/_Pair.TcPOU
FUNCTION INTERNAL _Pair : Result
VAR_INPUT
	iSignal		: I_SignalNode;
	iReceiver	: I_ReceiverNode;
END_VAR
VAR
	i			: UDINT;
	_nStart		: UDINT;
	_nEnd		: UDINT;
	_nFirstId	: UDINT;
	_nNextId	: UDINT;
	_nNewSize	: UDINT;
	_nNewStart	: UDINT;
END_VAR

// 1) Check if either iSignal or iReceiver is invalid (0 indicates null).
IF iSignal = 0 OR iReceiver = 0 THEN
	_Pair := Err.Itf0;
	RETURN;
END_IF

// 2) Check if global capacity is already at maximum.
IF _Broadcast.nRecLen = Param.RECEIVER_CAP THEN
	_Pair := Err.Ovf;
	RETURN;
END_IF

// 3) Ensure this exact iReceiver isn't already within the iSignal chunk
FOR i := iSignal._Start + 1 TO iSignal._End DO
	IF _Broadcast.entry[i].variant.iReceiver = iReceiver THEN
		_Pair := Err.ItfEq;
		RETURN;
	END_IF
END_FOR

// 4) If the signal is brand-new (_Start=0), try allocating exactly 2 slots.
IF iSignal._Start = 0 THEN
	CASE (_Pair := _BroadcastGetBestFit(2, nStart => _nStart, nEnd => _nEnd)) OF
		Ok:
			// Found a free chunk of size 2
		None:
			CASE (_Pair := _BroadcastDefragment()) OF 
				Ok:
					// We can safely assume that if _BroadcastGetBestFit and _BroadcastDefragment didn't failed then _Broadcast.nRecLen + 1 is the next unoccupied slot.
					// If _BroadcastGetBestFit failed then there is no avaliable space in the first place.
					// If _BroadcastDefragment failed then this wouldn't be executed.
					_nStart := _Broadcast.nRecLen + 1;
					_nEnd := _Broadcast.nRecLen + 2;
				ELSE
					RETURN;
			END_CASE
		ELSE
			// Any other error, just return
			RETURN;
	END_CASE

	IF IsOk(_Pair) THEN
		// Mark the first slot as signal header
		_Broadcast.entry[_nStart].nType := 1;
		_Broadcast.entry[_nStart].variant.iSignal := iSignal;

		// Mark the second slot as the receiver
		_Broadcast.entry[_nEnd].nType := 2;
		_Broadcast.entry[_nEnd].variant.iReceiver := iReceiver;

		// Update the signal's metadata
		iSignal._Start := _nStart;
		iSignal._End   := _nEnd;
		iSignal._Size := 2;

		// Increase global count of used slots
		_Broadcast.nRecLen := _Broadcast.nRecLen + 2;

		// Update _Broadcast.iFirst if needed
		IF _Broadcast.iFirst = 0 THEN
			_Broadcast.iFirst := iSignal;
		ELSIF iSignal._Start < _Broadcast.iFirst._Start THEN
			_Broadcast.iFirst := iSignal;
		END_IF

		RETURN;
	ELSE
		RETURN;
	END_IF
END_IF

// 5) If the signal already has slots, try extending to the right by 1 slot.
_nNextId := iSignal._End + 1;
IF (_nNextId <= Param.RECEIVER_CAP) AND_THEN (_Broadcast.entry[_nNextId].nType = 0) THEN
	// Mark that free slot as a new receiver
	_Broadcast.entry[_nNextId].nType := 2;
	_Broadcast.entry[_nNextId].variant.iReceiver := iReceiver;

	// Update signal info
	iSignal._End := _nNextId;
	iSignal._Size := iSignal._Size + 1;

	// Increase global used-slot counter
	_Broadcast.nRecLen := _Broadcast.nRecLen + 1;

	_Pair := Ok;
	RETURN;
END_IF

// 6) Try expanding to the left by shifting the boundary marker left one slot.
_nNextId := iSignal._Start - 1;
IF (_nNextId > 0) AND_THEN (_Broadcast.entry[_nNextId].nType = 0) THEN
	// Copy old boundary marker to new index
	_Broadcast.entry[_nNextId] := _Broadcast.entry[iSignal._Start];

	// Turn the old boundary marker slot into the new receiver
	_Broadcast.entry[iSignal._Start].nType := 2;
	_Broadcast.entry[iSignal._Start].variant.iReceiver := iReceiver;

	// Update signal to reflect new _Start
	iSignal._Start := _nNextId;
	iSignal._Size := iSignal._Size + 1;

	// Increase global used-slot counter
	_Broadcast.nRecLen := _Broadcast.nRecLen + 1;

	_Pair := Ok;
	RETURN;
END_IF

// 7) If neither immediate left nor right expansions are possible, we need a new chunk
_nNewSize := iSignal._Size + 1;
CASE (_Pair := _BroadcastGetBestFit(_nNewSize, nStart => _nStart, nEnd => _nEnd)) OF
	Ok:
		// Chunk found
	None:
		// No chunk found => defragment.
		CASE (_Pair := _BroadcastDefragment(iSignal)) OF 
			Ok:
				// As above
				_nStart := _Broadcast.nRecLen + 1;
				_nEnd := _Broadcast.nRecLen + _nNewSize;
			ELSE
				RETURN;
		END_CASE
	ELSE
		// Other errors
		RETURN;
END_CASE

IF IsOk(_Pair) THEN

	// Move the entire existing block to the new chunk
	Tc2_SYSTEM.MEMMOVE(
		ADR(_Broadcast.entry[_nStart]),
		ADR(_Broadcast.entry[iSignal._Start]),
		SIZEOF(_BroadcastStruct) * iSignal._Size
	);

	// Clear out the old region
	Tc2_SYSTEM.MEMSET(
		ADR(_Broadcast.entry[iSignal._Start]),
		0,
		SIZEOF(_BroadcastStruct) * iSignal._Size
	);

	// Mark the final slot in the new chunk as the new receiver
	_Broadcast.entry[_nEnd].nType := 2;
	_Broadcast.entry[_nEnd].variant.iReceiver := iReceiver;

	// Update the signal to reflect the new block location
	iSignal._Start := _nStart;
	iSignal._End   := _nEnd;
	iSignal._Size := iSignal._Size + 1;

	// One more slot used
	_Broadcast.nRecLen := _Broadcast.nRecLen + 1;

	// If this signal was iFirst, re-scan for the new leftmost. 
	// Otherwise, if we are now to the left of iFirst, update iFirst.
	IF _Broadcast.iFirst = iSignal THEN
		FOR i := 1 TO _Broadcast.nSignalLen DO
			_nNewStart := _Broadcast.iSignal[i]._Start;
			IF _nNewStart <> 0 AND_THEN _nNewStart < _nFirstId THEN
				_nFirstId := _Broadcast.iSignal[i]._Start;
				_Broadcast.iFirst := _Broadcast.iSignal[i];
			END_IF
		END_FOR
	ELSIF iSignal._Start < _Broadcast.iFirst._Start THEN
		_Broadcast.iFirst := iSignal;
	END_IF
END_IF

END_FUNCTION

// ---- Broadcast/Sys/Helpers/_BroadcastDefragment.TcPOU
FUNCTION INTERNAL _BroadcastDefragment : Result
VAR_INPUT
	iLastSignal		: I_SignalNode := 0;
END_VAR
VAR
	i				: UDINT;
   _temp			: ARRAY[1..Param.RECEIVER_CAP] OF _BroadcastStruct;
   _iSwappedSignal	: I_SignalNode;
   _nNextCopyId		: UDINT := 1;
END_VAR

// 1) If we are at maximum capacity (all slots are allocated).
IF _Broadcast.nRecLen = Param.RECEIVER_CAP THEN
    _BroadcastDefragment := Err.Ovf;
    RETURN;
END_IF

// 2) If there are no allocated slots at all, nothing to defragment.
IF _Broadcast.nRecLen = 0 THEN
    _BroadcastDefragment := Ok;
    RETURN;
END_IF

// 3) We want to ensure that entity that requires more space will get it, so we move it temporarly to the end.
IF iLastSignal <> 0 THEN
	_iSwappedSignal := _Broadcast.iSignal[_Broadcast.nSignalLen];
	_Broadcast.iSignal[iLastSignal._Id] := _iSwappedSignal;
	_Broadcast.iSignal[_Broadcast.nSignalLen] := iLastSignal;
END_IF

// 3) Copy all chunks to the temporary table
FOR i := 1 TO _Broadcast.nSignalLen DO
	IF _Broadcast.iSignal[i]._Start <> 0 THEN
		Tc2_SYSTEM.MEMCPY(
							ADR(_temp[_nNextCopyId]),
							ADR(_Broadcast.entry[_Broadcast.iSignal[i]._Start]),
							SIZEOF(_BroadcastStruct) * _Broadcast.iSignal[i]._Size
						);
		_Broadcast.iSignal[i]._Start := _nNextCopyId;
		_nNextCopyId := _Broadcast.iSignal[i]._Size + _nNextCopyId;
		_Broadcast.iSignal[i]._End := _nNextCopyId - 1;	
	END_IF
END_FOR

// 3) Move back the swapped entities, to preserve the Ids.
IF iLastSignal <> 0 THEN
	_Broadcast.iSignal[_iSwappedSignal._Id] := _iSwappedSignal;
	_Broadcast.iSignal[iLastSignal._Id] := iLastSignal;
END_IF

// 4) Copy temporary table onto the _Ec.comp table
Tc2_System.MEMCPY(
	ADR(_Broadcast.entry),
	ADR(_temp),
	SIZEOF(_BroadcastStruct) * _Broadcast.nRecLen
);

// 5) Clear the remainging area
Tc2_System.MEMSET(
	ADR(_Broadcast.entry[_Broadcast.nRecLen + 1]),
	0,
	SIZEOF(_BroadcastStruct) * (Param.RECEIVER_CAP - _Broadcast.nRecLen)
);

// 6) First entry in _Ec.comp should always be iFirst
CASE _Broadcast.entry[1].nType OF
	1:
		_BroadcastDefragment := Ok;
		_Broadcast.iFirst := _Broadcast.entry[1].variant.iSignal;
	ELSE
		_BroadcastDefragment := Err.Udf;
END_CASE

END_FUNCTION

// ---- Result/IsOk.TcPOU
// Return TRUE on a successful (Ok) result.
// Optionally carries the value over to nOut for further processing.
FUNCTION IsOk : BOOL
VAR_INPUT
    nIn : Result; // Result variable to check for success
END_VAR
VAR_OUTPUT
    nOut : Result; // Carries the input value for further use
END_VAR

IsOk := nIn > 0;
nOut := nIn;

END_FUNCTION

// ---- Broadcast/Receiver/Receiver.TcPOU
(*
Represents a receiver in the Broadcast system. Implements the necessary methods for receiving events and pairing signals.
*)
FUNCTION_BLOCK Receiver IMPLEMENTS I_Receiver, I_Callable
VAR
	{ attribute 'hide' }
	_comp: Component(THIS^);

	{ attribute 'hide' }
	_iCallable: I_Callable := THIS^;
	
	_tag: TagBase;
END_VAR

(*
This method provides a standardized way for other objects to interact with the object that owns it.
*)
{ attribute 'hide' }
METHOD Call
VAR_INPUT
	iArg	: I_Arg;
END_VAR
END_METHOD

PROPERTY FINAL Callable : I_Callable
GET
Callable := _iCallable;
END_GET
SET
_iCallable := Callable;
END_SET
END_PROPERTY

METHOD INTERNAL Receive
VAR_INPUT
	iArg			: I_Arg;
END_VAR
IF _iCallable = 0 THEN
	NewDebug(THIS^, Param.EXE_INTERNAL_DEBUG_MODE, 'Callable = 0!');
	RETURN;
END_IF

_iCallable.Call(iArg);
END_METHOD

(*
Provides access to the tag associated with the signal.
*)
PROPERTY FINAL Tag : I_Tag
GET
Tag := _tag;
END_GET
END_PROPERTY

END_FUNCTION_BLOCK

// ---- Runtime/Runtime.TcPOU
(*
Manages the initialization and cyclic execution of registered function blocks.
*)
FUNCTION Runtime
VAR
	iInit: I_InitNode := _Runtime.iFirstInit;
	iExecute: I_ExecuteNode := _Runtime.iFirstCyclic;
END_VAR

IF _Runtime.bInit THEN
	WHILE iInit <> 0 DO
		iInit.Init(iNext => iInit);
	END_WHILE

	IF _Ec.nConstructedScopes <> 0 THEN
		NewDebug(0, Param.INIT_INTERNAL_DEBUG_MODE, 'Close all Entity scopes!');
	END_IF
	
	IF _Debug.nPanicNumber > 0 THEN
		_Runtime.iFirstCyclic := 0;
		Tc2_System.ADSLOGSTR(Tc2_System.ADSLOG_MSGTYPE_ERROR, Tc2_Standard.CONCAT('Runtime disabled! Debug panics: ', UDINT_TO_STRING(_Debug.nPanicNumber)), '');
	END_IF
	
	IF _Debug.nNotifyNumber > 0 THEN
		_Runtime.iFirstCyclic := 0;
		Tc2_System.ADSLOGSTR(Tc2_System.ADSLOG_MSGTYPE_WARN, Tc2_Standard.CONCAT('Debug notifies: ', UDINT_TO_STRING(_Debug.nPanicNumber)), '');
	END_IF
	
	_Runtime.bInit := FALSE;
END_IF

WHILE iExecute <> 0 DO
	iExecute.Exe(iNext => iExecute);
END_WHILE

END_FUNCTION

// ---- Broadcast/Arg/IArgToIComp.TcPOU
(*
Casts I_Arg as I_Component.
Returns:
- Ok - Success,
- Err.InvRef - Invalid reference,
- Err.Itf0 - Invalid interface,
- Err.NoMatch - Cast failed
*)
FUNCTION IArgToIComp : Result
VAR_INPUT
	iIn		: I_Arg;
	iOut	: REFERENCE TO I_RawComponent;
END_VAR

IF NOT __ISVALIDREF(iOut) THEN
	IArgToIComp := Err.InvRef;
	RETURN;
END_IF

IF iIn = 0 THEN
	IArgToIComp := Err.Itf0;
	RETURN;
END_IF

IF __QUERYINTERFACE(iIn, iOut) THEN
	IArgToIComp := Ok;
ELSE
	IArgToIComp := Err.NoMatch;
END_IF

END_FUNCTION

// ---- Broadcast/Helpers/GetReceiver.TcPOU
(*
Searches an `I_Entity` for a `I_Receiver` component matching provided id pattern.
Result:
- Ok - Returns `I_Receiver`.
- Err.NotFound - Returns null.
- Err.InvRef - Returns null.
- Err.Itf0 - Returns null, incorrect interface.
*)
FUNCTION GetReceiver : Result
VAR_INPUT
	iEntity		: I_Entity;
	sTagId		: Str;
	iOut		: REFERENCE TO I_Receiver;
END_VAR
VAR
	_iComp		: I_Component;
	cmp			: TagCmp;
END_VAR

IF iEntity = 0 THEN
	GetReceiver := Err.Itf0;
	RETURN;
END_IF

IF NOT __ISVALIDREF(iOut) THEN
	GetReceiver := Err.InvRef;
	RETURN;
END_IF

WHILE IsOk(iEntity.GetNextComp(_iComp)) DO
	IF IsOk(ICompToIRec(_iComp.Raw, iOut)) THEN
		IF cmp.Set(iOut.Tag).MatchWcdId(sTagId).IsTrue() THEN
			GetReceiver := Ok;
			RETURN;
		ELSE
			iOut := 0;
		END_IF
	END_IF
END_WHILE

GetReceiver := Err.NotFound;

END_FUNCTION

// ---- Broadcast/Signal/ICompToISignal.TcPOU
(*
Casts I_Component as I_Signal.
Returns:
- Ok - Success,
- Err.InvRef - Invalid reference,
- Err.Itf0 - Invalid interface,
- Err.NoMatch - Cast failed
*)
FUNCTION ICompToISignal : Result
VAR_INPUT
	iIn	: I_RawComponent;
	iOut: REFERENCE TO I_Signal;
END_VAR

IF NOT __ISVALIDREF(iOut) THEN
	ICompToISignal := Err.InvRef;
	RETURN;
END_IF

IF iIn = 0 THEN
	ICompToISignal := Err.Itf0;
	RETURN;
END_IF

IF __QUERYINTERFACE(iIn, iOut) THEN
	ICompToISignal := Ok;
ELSE
	ICompToISignal := Err.NoMatch;
END_IF

END_FUNCTION

// ---- Dbg/DebugInfo.TcPOU
(*
Provides access to registered debug information, enabling monitoring and troubleshooting of system components.
*)
FUNCTION_BLOCK DebugInfo
VAR
	nLastMsgIdx: REFERENCE TO UDINT REF= _Debug.nLastIdx;
	nTotalNumber: REFERENCE TO UDINT REF= _Debug.nTotalNumber;
	nPanicNumber: REFERENCE TO UDINT REF= _Debug.nPanicNumber;
	nNotifyNumber: REFERENCE TO UDINT REF= _Debug.nNotifyNumber;
	entry: REFERENCE TO ARRAY[1..Param.DEBUG_CAP] OF _DebugInfo REF= _Debug.debugMsg;	
END_VAR

END_FUNCTION_BLOCK

// ---- Entity/Core/Scope/EntityEnd.TcPOU
(*
Defines end of an entity scope outside which no new component can be registered.
*)
FUNCTION_BLOCK EntityEnd IMPLEMENTS I_Debug

//FB_Init is always available implicitly and it is used primarily for initialization.
//The return value is not evaluated. For a specific influence, you can also declare the
//methods explicitly and provide additional code there with the standard initialization
//code. You can evaluate the return value.
{attribute 'hide'}
METHOD FB_Init: BOOL
VAR_INPUT
    bInitRetains: BOOL; // TRUE: the retain variables are initialized (reset warm / reset cold)
    bInCopyCode: BOOL;  // TRUE: the instance will be copied to the copy code afterward (online change)   
END_VAR
VAR
	_nResult	: Result;
END_VAR
IF IsErr(_EntityEnd(), nOut => _nResult) THEN
	NewDebug(THIS^, Param.INIT_INTERNAL_DEBUG_MODE, Tc2_Standard.CONCAT('EndEntity() failed with code: ', ResultToStr(_nResult)));
END_IF
END_METHOD

END_FUNCTION_BLOCK

// ---- Entity/Sys/_Helpers/_EntityEnd.TcPOU
FUNCTION INTERNAL _EntityEnd : Result
VAR
	iEntity: I_Entity;
END_VAR

// Check if the runtime system is initialized
IF NOT _Runtime.bInit THEN
    // If not initialized, return with an initialization error
    _EntityEnd := Err.Init;
    RETURN;
END_IF

// Check if there is an entity currently under construction
IF _Ec.iUnderConstruction = 0 THEN
    // If no entity is under construction, return with interface error
    _EntityEnd := Err.Itf0;
    RETURN;
END_IF

// Mark the current under-construction entity as completed
_Ec.iUnderConstruction._State := _EntityState.Completed;

// Decrement the count of constructed scopes
_Ec.nConstructedScopes := _Ec.nConstructedScopes - 1;

// If there are still scopes left to complete
IF _Ec.nConstructedScopes > 0 THEN
    // Traverse backwards to find an entity that is registered but not yet completed
	iEntity := _Ec.iUnderConstruction;
    WHILE IsOk(GetPrevEntity(iEntity)) DO
        // If a registered entity is found, set the return value to OK and exit
        IF _Ec.iUnderConstruction._State = _EntityState.Registered THEN
            _EntityEnd := Ok;
            RETURN;
        END_IF
    END_WHILE

    // If all remaining entities are completed, reset under-construction pointer and return OK
    _Ec.iUnderConstruction := 0;
    _EntityEnd := Ok;
ELSE
    // If no scopes left, reset under-construction pointer and return OK
    _Ec.iUnderConstruction := 0;
    _EntityEnd := Ok;
END_IF

END_FUNCTION

// ---- Entity/Core/GetPrevEntity.TcPOU
(*
Retrieves the I_Entity instance. It is either previous entity in relation to the inputted one or last entity if passed interface pointer contains null.

Results:
- Ok - Success. Replaces value of iEntity with the last or previous entity.
- Err.InvRef - Invalid reference.
- Err.Itf0 - No entity. Nulls passed interface pointer.
- Err.End - End of collection. Nulls passed interface pointer.
*)
FUNCTION GetPrevEntity : Result
VAR_INPUT
	iEntity: REFERENCE TO I_Entity;
END_VAR
VAR
END_VAR

// Check if the given entity reference is valid
IF NOT __ISVALIDREF(iEntity) THEN
    // If the reference is invalid, return with an invalid reference error
    GetPrevEntity := Err.InvRef;
    RETURN;
END_IF

// Check if the entity chain has been initialized (i.e., if there's a last entity)
IF _Ec.iLast = 0 THEN
    // If not initialized, return with interface error
	iEntity := 0;
    GetPrevEntity := Err.Itf0;
    RETURN;
END_IF

// If input entity is 0, start iteration from the last entity in the list
IF iEntity = 0 THEN
    iEntity := _Ec.iLast;
    GetPrevEntity := Ok;

// If the current entity has a previous one, move to it
ELSIF iEntity._Prev <> 0 THEN
    iEntity := iEntity._Prev;
    GetPrevEntity := Ok;

// If there is no previous entity, beginning of the list is reached
ELSE
	iEntity := 0;
    GetPrevEntity := Err.End;
END_IF

END_FUNCTION

// ---- Entity/Core/Scope/EntityExtend.TcPOU
(*
Reopens an entity scope for modifications.
*)
FUNCTION_BLOCK EntityExtend IMPLEMENTS I_Debug

//FB_Init is always available implicitly and it is used primarily for initialization.
//The return value is not evaluated. For a specific influence, you can also declare the
//methods explicitly and provide additional code there with the standard initialization
//code. You can evaluate the return value.
{attribute 'hide'}
METHOD FB_Init: BOOL
VAR_INPUT
    bInitRetains: BOOL; // TRUE: the retain variables are initialized (reset warm / reset cold)
    bInCopyCode: BOOL;  // TRUE: the instance will be copied to the copy code afterward (online change)
	
	iEntity	: I_Entity;
END_VAR
VAR
	_nResult	: Result;
END_VAR
IF IsErr(_EntityExtend(iEntity), nOut => _nResult) THEN
	NewDebug(THIS^, Param.INIT_INTERNAL_DEBUG_MODE, Tc2_Standard.CONCAT('ExtendEntity(I_EntityNode) failed with code: ', ResultToStr(_nResult)));
END_IF
END_METHOD

END_FUNCTION_BLOCK

// ---- Entity/Core/Scope/EntityStart.TcPOU
(*
Represents a registered entity in the Entity-Component system and start of its scope.
Nested scopes are possible, components are always registered within most inner scope.
*)
FUNCTION_BLOCK EntityStart IMPLEMENTS I_Entity, I_Debug;
VAR
	_eState: _EntityState;
	_iNext: I_Entity;
	_iPrev: I_Entity;
	_iFirstComp: I_Component;
	_iLastComp: I_Component;
	_nSize: UDINT;
END_VAR

PROPERTY INTERNAL _FirstComp : I_Component
GET
_FirstComp := _iFirstComp;
END_GET
SET
_iFirstComp := _FirstComp;
END_SET
END_PROPERTY

PROPERTY INTERNAL _LastComp : I_Component
GET
_LastComp := _iLastComp;
END_GET
SET
_iLastComp := _LastComp;
END_SET
END_PROPERTY

PROPERTY INTERNAL _Next : I_Entity
GET
_Next := _iNext;
END_GET
SET
_iNext := _Next;
END_SET
END_PROPERTY

PROPERTY INTERNAL _Prev : I_Entity
GET
_Prev := _iPrev;
END_GET
SET
_iPrev := _Prev;
END_SET
END_PROPERTY

PROPERTY INTERNAL _Size : UDINT
GET
_Size := _nSize;
END_GET
SET
_nSize := _Size;
END_SET
END_PROPERTY

PROPERTY INTERNAL _State : _EntityState
GET
_State := _eState;
END_GET
SET
_eState := _State;
END_SET
END_PROPERTY

//FB_Init is always available implicitly and it is used primarily for initialization.
//The return value is not evaluated. For a specific influence, you can also declare the
//methods explicitly and provide additional code there with the standard initialization
//code. You can evaluate the return value.
{attribute 'hide'}
METHOD FB_Init: BOOL
VAR_INPUT
    bInitRetains: BOOL; // TRUE: the retain variables are initialized (reset warm / reset cold)
    bInCopyCode: BOOL;  // TRUE: the instance will be copied to the copy code afterward (online change)
END_VAR
VAR
	_nResult	: Result;
END_VAR
IF IsErr(_EntityStart(THIS^), nOut => _nResult) THEN
	NewDebug(THIS^, Param.INIT_INTERNAL_DEBUG_MODE, Tc2_Standard.CONCAT('_StartEntity(THIS^) failed with code: ', ResultToStr(_nResult)));
END_IF
END_METHOD

(*
Description: Retrieves a next component after the inputted one or first component if referenced value is 0. 
Returns:
- Ok - Returns upon success, updates referenced value with new component.
- Err.InvRef - Invalid output reference.
- Err.ItfEq - Provided interface pointer doesn't belong to the queried entity. Nulls reference.
- Err.NotFound - The entity doesn't contain any components. Nulls reference.
- Err.End - No more components. Nulls reference.
*)
METHOD GetNextComp : Result
VAR_INPUT
	iOut	: REFERENCE TO I_Component;
END_VAR
VAR
	_iThis: I_Entity := THIS^;
END_VAR
// Check if the given output reference is valid
IF NOT __ISVALIDREF(iOut) THEN
    // If not a valid reference, return invalid reference error
    GetNextComp := Err.InvRef;
    RETURN;
END_IF

// If no starting component is specified, begin with the first component
IF iOut = 0 THEN
    IF _iFirstComp <> 0 THEN
        // Return the first component in the list
        iOut := _iFirstComp;
        GetNextComp := Ok;
    ELSE
        // No components exist in the list
        GetNextComp := Err.NotFound;
    END_IF

// If the current component does not belong to this entity, reject the call
ELSIF iOut._Entity <> _iThis THEN
    // Cross-linked or stale reference: component doesn't belong to this context
	iOut := 0;
    GetNextComp := Err.ItfEq;

// If there's no next component, we've reached the end of the list
ELSIF iOut._Next = 0 THEN
	iOut := 0;
    GetNextComp := Err.End;

// Otherwise, return the next component in the list
ELSE
    iOut := iOut._Next;
    GetNextComp := Ok;
END_IF
END_METHOD

(*
Description: Retrieves a previous component before the inputted one or last component if referenced value is 0.
Returns:
- Ok - Returns upon success, updates referenced value with new component.
- Err.InvRef - Invalid output reference.
- Err.ItfEq - Provided interface pointer doesn't belong to the queried entity. Nulls reference.
- Err.NotFound - The entity doesn't contain any components. Nulls reference.
- Err.End - No more components. Nulls reference.
*)
METHOD GetPrevComp : Result
VAR_INPUT
	iOut	: REFERENCE TO I_Component;
END_VAR
VAR
	_iThis: I_Entity := THIS^;
END_VAR
// Check if the given output reference is valid
IF NOT __ISVALIDREF(iOut) THEN
    // If not a valid reference, return invalid reference error
    GetPrevComp := Err.InvRef;
    RETURN;
END_IF

// If no starting component is specified, begin with the first component
IF iOut = 0 THEN
    IF _iLastComp <> 0 THEN
        // Return the first component in the list
        iOut := _iLastComp;
        GetPrevComp := Ok;
    ELSE
        // No components exist in the list
        GetPrevComp := Err.NotFound;
    END_IF

// If the current component does not belong to this entity, reject the call
ELSIF iOut._Entity <> _iThis THEN
    // Cross-linked or stale reference: component doesn't belong to this context
	iOut := 0;
    GetPrevComp := Err.ItfEq;

// If there's no next component, we've reached the end of the list
ELSIF iOut._Prev = 0 THEN
	iOut := 0;
    GetPrevComp := Err.End;

// Otherwise, return the next component in the list
ELSE
    iOut := iOut._Prev;
    GetPrevComp := Ok;
END_IF
END_METHOD

(*
Provides the size of the entity, indicating the number of components it manages.  
Note: For internal logic purposes, this value is incremented by one beyond the actual component count.
*)
PROPERTY Size : UDINT
GET
Size := _nSize;
END_GET
END_PROPERTY

END_FUNCTION_BLOCK

// ---- Entity/Core/GetOwnerFromRaw.TcPOU
(*
Finds the owning entity of a given component in the Entity-Component system.  
This function may involve a costly search operation, iterating through all components.
Returns:
- `Ok` - Successfully retrieves the `I_Entity` that owns the component.
- `Err.Itf0` - iIn = 0.
- `Err.InvRef` - Invalid output reference.
- `Err.NotFound` - No owning entity is found, returning null.
*)
FUNCTION GetOwnerFromRaw : Result
VAR_INPUT
	iIn: I_RawComponent;
	iOut: REFERENCE TO I_Entity;
END_VAR
VAR
	_iComp		: I_Component;
END_VAR

IF iIn = 0 THEN
	GetOwnerFromRaw := Err.Itf0;
	RETURN;
END_IF

IF NOT __ISVALIDREF(iOut) THEN
	GetOwnerFromRaw := Err.InvRef;
	RETURN;
END_IF

WHILE IsOk(GetNextEntity(iOut)) DO
	WHILE IsOk(iOut.GetNextComp(_iComp)) DO
		IF _iComp.Raw = iIn THEN
			GetOwnerFromRaw := Ok;
			RETURN;
		END_IF
	END_WHILE
END_WHILE

GetOwnerFromRaw := Err.NotFound;

END_FUNCTION

// ---- Entity/Core/GetNextEntity.TcPOU
(*
Retrieves the I_Entity instance. It is either next entity in relation to the inputted one or first entity if passed interface pointer contains null.

Results:
- Ok - Success. Replaces value of iEntity with the first or following entity.
- Err.InvRef - Invalid reference.
- Err.Itf0 - No entity. Nulls passed interface pointer.
- Err.End - End of collection. Nulls passed interface pointer.
*)
FUNCTION GetNextEntity : Result
VAR_INPUT
	iEntity: REFERENCE TO I_Entity;
END_VAR
VAR
END_VAR

// Check if the given entity reference is valid
IF NOT __ISVALIDREF(iEntity) THEN
    // If the reference is invalid, return with an invalid reference error
    GetNextEntity := Err.InvRef;
    RETURN;
END_IF

// Check if the entity chain has been initialized (i.e., if there's a first entity)
IF _Ec.iFirst = 0 THEN
    // If not initialized, return with interface error
	iEntity := 0;
    GetNextEntity := Err.Itf0;
    RETURN;
END_IF

// If input entity is 0, start iteration from the first entity in the list
IF iEntity = 0 THEN
    iEntity := _Ec.iFirst;
    GetNextEntity := Ok;

// If the current entity has a next one, move to it
ELSIF iEntity._Next <> 0 THEN
    iEntity := iEntity._Next;
    GetNextEntity := Ok;

// If there is no next entity, end of the list is reached
ELSE
    iEntity := 0;
    GetNextEntity := Err.End;
END_IF

END_FUNCTION

// ---- Result/IsFail.TcPOU
// Return TRUE on a NON successful (NOT Ok) result.
// Optionally carries the value over to nOut for further processing.
FUNCTION IsFail : BOOL
VAR_INPUT
    nIn : Result; // Result variable to check for success
END_VAR
VAR_OUTPUT
    nOut : Result; // Carries the input value for further use
END_VAR

IsFail := nIn <= 0;
nOut := nIn;

END_FUNCTION

// ---- Result/IsEnd.TcPOU
// Return TRUE for nIn = Err.End.
// Optionally carries the value over to nOut for further processing.
FUNCTION IsEnd : BOOL
VAR_INPUT
    nIn : Result; // Result variable to check for any non-None value
END_VAR
VAR_OUTPUT
    nOut : Result; // Carries the input value for further use
END_VAR

IsEnd := nIn = Err.End;
nOut := nIn;

END_FUNCTION

// ---- Runtime/Execute/Execute.TcPOU
(*
Allows registration of FB implementing `I_Execute`. 
*)
FUNCTION_BLOCK FINAL Execute IMPLEMENTS I_ExecuteNode, I_Debug
VAR
	_iExecute		: I_Execute;
	_iNext			: I_ExecuteNode;
	_nState			: Result;
	_nPhase			: INT;
END_VAR

METHOD INTERNAL Attach : Result
VAR_INPUT
	iExecute		: I_ExecuteNode;
END_VAR
VAR
	_iThis			: I_ExecuteNode := THIS^;
END_VAR
IF iExecute = 0 THEN
	NewDebug(THIS^, Param.INIT_INTERNAL_DEBUG_MODE, Tc2_Standard.CONCAT(__POUNAME(), ': Itf = 0!'));
	RETURN;
END_IF

IF _iThis <> _Runtime.iLastCyclic THEN
	NewDebug(THIS^, Param.INIT_INTERNAL_DEBUG_MODE, Tc2_Standard.CONCAT(__POUNAME(), ': Is not the last node!'));
	RETURN;
END_IF

IF IsSome(iExecute.state) THEN
	NewDebug(iExecute, Param.INIT_INTERNAL_DEBUG_MODE, Tc2_Standard.CONCAT(__POUNAME(), ': Has already been added!'));
	RETURN;
END_IF

_Runtime.iLastCyclic := iExecute;
_iNext := iExecute;
END_METHOD

METHOD INTERNAL Exe
VAR_OUTPUT
	iNext: I_ExecuteNode;
END_VAR
_iExecute.Execute(_nPhase);
iNext := _iNext;
END_METHOD

//FB_Init is always available implicitly and it is used primarily for initialization.
//The return value is not evaluated. For a specific influence, you can also declare the
//methods explicitly and provide additional code there with the standard initialization
//code. You can evaluate the return value.
{attribute 'hide'}
METHOD FB_Init: BOOL
VAR_INPUT
    bInitRetains: BOOL; // TRUE: the retain variables are initialized (reset warm / reset cold)
    bInCopyCode: BOOL;  // TRUE: the instance will be copied to the copy code afterward (online change)
	
	iExecute			: I_Execute;
END_VAR
IF IsSome(_nState) THEN
	RETURN;
END_IF

IF (_iExecute := iExecute) = 0 THEN
	_nState := Err.Itf0;
	NewDebug(THIS^, Param.INIT_INTERNAL_DEBUG_MODE, Tc2_Standard.CONCAT(__POUNAME(), ': Itf = 0!'));
	RETURN;
END_IF



IF _Runtime.iLastCyclic <> 0 THEN
	IF IsErr(_Runtime.iLastCyclic.Attach(THIS^), nOut => _nState) THEN
		NewDebug(THIS^, Param.INIT_INTERNAL_DEBUG_MODE, Tc2_Standard.CONCAT(__POUNAME(), ': Error Inside!'));
	END_IF
ELSE
	_Runtime.iFirstCyclic := THIS^;
	_Runtime.iLastCyclic := THIS^;
	_nState := Ok;
END_IF
END_METHOD

PROPERTY Phase : INT
GET
Phase := _nPhase;
END_GET
SET
_nPhase := Phase;
END_SET
END_PROPERTY

PROPERTY INTERNAL State : Result
GET
State := _nState;
END_GET
SET
IF IsNone(_nState) THEN
	_nState := State;
END_IF
END_SET
END_PROPERTY

END_FUNCTION_BLOCK

// ---- State/_Buffer/_StateBuffer.TcPOU
(*
A buffer for storing states.  
*)
FUNCTION_BLOCK INTERNAL _StateBuffer
VAR
	_iFirst				: I_State;
	_iLast				: I_State;
	_nLen				: UDINT;
END_VAR

(*
Returns the current number of states stored in the buffer.
*)
METHOD Length : UDINT
VAR_INPUT
END_VAR
Length := _nLen;
END_METHOD

(*
Removes and retrieves the oldest state from the buffer.  

Returns:
- `Ok` - If a state is successfully removed.
- `None` - If the buffer is empty.
*)
METHOD Pop : Result
VAR_OUTPUT
	iState			: I_State;
END_VAR
IF _iFirst = 0 THEN
	Pop := None;
	RETURN;
END_IF

iState := _iFirst;
_iFirst := _iFirst._NextInBuffer;
iState._NextInBuffer := 0;
iState._InQueue := FALSE;

IF _iFirst = 0 THEN
	_iLast := 0;
END_IF

_nLen := _nLen - 1;
Pop := Ok;
END_METHOD

(*
Adds a new state to the buffer.  
Returns:
- `Ok` - If the state is successfully added.
- `Err.Itf0` - If the provided state interface is invalid.
- `Err.IncArg` - Uf the provided state already is in some buffer.
*)
METHOD Push : Result
VAR_INPUT
	iState			: I_State;
END_VAR
IF iState = 0 THEN
	Push := Err.Itf0;
	RETURN;
END_IF

IF iState._InQueue THEN
	Push := Err.IncArg;
	RETURN;
END_IF

IF _iLast = 0 THEN
	_iFirst := iState;
	_iLast := iState;
	iState._InQueue := TRUE;
	_nLen := _nLen + 1;
ELSE
	_iLast._NextInBuffer := iState;
	_iLast := iState;
	iState._InQueue := TRUE;
	_nLen := _nLen + 1;
END_IF

Push := Ok;
END_METHOD

END_FUNCTION_BLOCK

// ---- State/Helpers/GetStateManager.TcPOU
(*
Searches an `I_Entity` for a `I_StateManager` component matching provided id pattern.
Result:
- Ok - Returns `I_StateManager`.
- Err.NotFound - Returns null.
- Err.InvRef - Returns null.
- Err.Itf0 - Returns null, incorrect interface.
*)
FUNCTION GetStateManager : Result
VAR_INPUT
	iEntity		: I_Entity;
	iOut		: REFERENCE TO I_StateManager;
END_VAR
VAR
	_iComp		: I_Component;
	cmp			: TagCmp;
END_VAR

IF iEntity = 0 THEN
	GetStateManager := Err.Itf0;
	RETURN;
END_IF

IF NOT __ISVALIDREF(iOut) THEN
	GetStateManager := Err.InvRef;
	RETURN;
END_IF

WHILE IsOk(iEntity.GetNextComp(_iComp)) DO
	IF IsOk(ICompToIStateMgr(_iComp.Raw, iOut)) THEN
		GetStateManager := Ok;
		RETURN;
	END_IF
END_WHILE

GetStateManager := Err.NotFound;

END_FUNCTION

// ---- State/Manager/ICompToIStateMgr.TcPOU
(*
Casts I_Component as I_StateManager.
Returns:
- Ok - Success,
- Err.InvRef - Invalid reference,
- Err.Itf0 - Invalid interface,
- Err.NoMatch - Cast failed
*)
FUNCTION ICompToIStateMgr : Result
VAR_INPUT
	iIn		: I_RawComponent;
	iOut	: REFERENCE TO I_StateManager;
END_VAR

IF NOT __ISVALIDREF(iOut) THEN
	ICompToIStateMgr := Err.InvRef;
	RETURN;
END_IF

IF iIn = 0 THEN
	ICompToIStateMgr := Err.Itf0;
	RETURN;
END_IF

IF __QUERYINTERFACE(iIn, iOut) THEN
	ICompToIStateMgr := Ok;
ELSE
	ICompToIStateMgr := Err.NoMatch;
END_IF

END_FUNCTION

// ---- State/_Machine/_StateMachine.TcPOU
FUNCTION_BLOCK INTERNAL _StateMachine IMPLEMENTS I_Execute
VAR
	_exe					: Execute(THIS^);
	_iCurrentState			: I_State;
END_VAR

(*
Changes the current state to a new state.  

Returns:
- `Ok` - If the state transition is successful.
- `Err.Itf0` - If the new state interface is invalid.
- `None` - If the transition cannot be completed due to state conditions.
*)
METHOD Change : Result
VAR_INPUT
	iNewState	: I_State;
END_VAR
VAR_OUTPUT
	iOldState	: I_State;
END_VAR
IF iNewState = 0 THEN
	Change := Err.Itf0;
	RETURN;
END_IF

IF iNewState = _iCurrentState THEN
	Change := None;
	RETURN;
END_IF

IF NOT iNewState._CanActivate() THEN
	Change := None;
	RETURN;
END_IF

IF _iCurrentState <> 0 AND_THEN NOT _iCurrentState._CanDeactivate() THEN
	Change := None;
	RETURN;
END_IF

IF _iCurrentState <> 0 THEN
	_iCurrentState._OnExit();
END_IF

iNewState._OnEntry();
iOldState := _iCurrentState;
_iCurrentState := iNewState;
Change := Ok;
END_METHOD

METHOD Execute
VAR_INPUT
	nPhase: INT := 0;
END_VAR
IF _iCurrentState <> 0 THEN
	_iCurrentState._OnExecute();
END_IF
END_METHOD

(*
Provides access to the current state, enabling inspection or external interaction with the state.
*)
PROPERTY State : I_State
GET
State := _iCurrentState;
END_GET
END_PROPERTY

END_FUNCTION_BLOCK

// ---- State/Manager/StateManager.TcPOU
(*
Manages the lifecycle and transitions of states within an entity.  
Supports queuing state change requests, triggering state transitions, and broadcasting state change events.  
Adds a `_stateChangeEvent` Signal to the owning `I_Entity` during initialization, enabling external components to listen for state changes.
*)
FUNCTION_BLOCK FINAL StateManager IMPLEMENTS I_Execute, I_StateManager, I_Debug

VAR
	_comp				: Component(THIS^);

	_exe				: Execute(THIS^);
	_sm					: _StateMachine;
	_buffer				: _StateBuffer;
	
	_stateChangeEvent	: Signal;
	
	_iPretender			: I_State;
	_iCurrent			: I_State;
	_iPrevious 			: I_State;
	
	
END_VAR

(*
Retrieves the currently active state managed by the state manager.
*)
PROPERTY Current : I_State
GET
Current := _iCurrent;
END_GET
END_PROPERTY

// DO NOT CALL MANUALLY
{attribute 'hide'}
METHOD Execute
VAR_INPUT
	nPhase: INT := 0;
END_VAR
VAR
	_iNewState		: I_State;
	_iOldState		: I_State;
END_VAR
IF IsOk(_buffer.Pop(iState => _iNewState)) THEN
	_iPretender := _iNewState;
	IF IsOk(_sm.Change(_iNewState, iOldState => _iOldState)) THEN
		_stateChangeEvent.Emit(_iNewState.Tag);
		
		_iCurrent		:= _iNewState;
		IF _iOldState <> 0 THEN
			_iPrevious		:= _iOldState;
		END_IF
		
	END_IF
	
	_iPretender		:= 0;
END_IF
END_METHOD

(*
Returns the entity that owns this state.
*)
PROPERTY Owner : I_Entity
GET
Owner := _comp.Entity;
END_GET
END_PROPERTY

(*
Retrieves the state that is queued to become active next, but has not yet transitioned.
*)
PROPERTY Pretender : I_State
GET
Pretender := _iPretender;
END_GET
END_PROPERTY

(*
Retrieves the last active state prior to the current one.
*)
PROPERTY Previous : I_State
GET
Previous := _iPrevious;
END_GET
END_PROPERTY

(*
Allows initializing an external interface variable with an interface pointer to this instance within declaration block.
Example:
iSMgr: I_StateManager;
smgr: StateManager := (Proxy := iSMgr);
Result: iSMgr <> 0 
*)
PROPERTY Proxy : REFERENCE TO I_StateManager
SET
Proxy := THIS^;
END_SET
END_PROPERTY

(*
Queues a request to transition to a specified state.  
Returns:
- `Ok` - If the state change request is successfully queued.
- `Err.Itf0` - If the provided state interface is invalid.
- `Err.NoMatch` - If the state does not belong to the same entity.
- `Err.IncArg` - If the state is already in the queue.
*)
METHOD Request : Result
VAR_INPUT
	iState			: I_State;
END_VAR
VAR
	iStateInternal	: I_StateInternal;
END_VAR
IF iState = 0 THEN
	Request := Err.Itf0;
	RETURN;
END_IF

IF iState.Owner <> _comp.Entity THEN
	Request := Err.NoMatch;
	RETURN;
END_IF

Request := _buffer.Push(iState);
END_METHOD

END_FUNCTION_BLOCK

// ---- Strings/Strb/Strb.TcPOU
// A string builder utility that allows for manipulation of a string up to 255 characters. It implements the I_Strb interface that allows for method chaining.
FUNCTION_BLOCK FINAL Strb IMPLEMENTS I_Strb
VAR
	_sString	: Str;
	_nLength	: INT;
END_VAR

PROPERTY PRIVATE _this : I_Strb
GET
VAR
	_iThis : I_Strb := THIS^;
END_VAR
_this := _iThis;
END_GET
END_PROPERTY

// Appends the specified string to the current string.
// Truncates if the total length exceeds 255 characters.
METHOD Append : I_Strb
VAR_INPUT
    sToAdd : Str; // String to append
END_VAR

VAR
	_nNewLength	: INT;
END_VAR
Append := _this;

IF sToAdd = '' THEN
	RETURN;
END_IF

_nNewLength := Tc2_Standard.LEN(sToAdd) + _nLength;
IF _nNewLength > 255 THEN
	_nNewLength := 255;
END_IF

_sString := Tc2_Standard.CONCAT(_sString, sToAdd);
_nLength := _nNewLength;
END_METHOD

// Finds the first occurrence of a substring after the specified position.
// Outputs the start and end positions of the found substring.
METHOD FindFirstAfter : I_Strb
VAR_INPUT
    sToFind : Str;      // Substring to find
    nPosition : INT := 1; // Starting position for search
END_VAR
VAR_OUTPUT
    nStart : INT;       // Start position of the found substring
    nEnd : INT;         // End position of the found substring
END_VAR

VAR
	_sTemp			: Str;
	_nOffset		: INT;
END_VAR
FindFirstAfter := _this;

IF sToFind = '' THEN
	RETURN;
END_IF

IF nPosition = 0 THEN
	RETURN;
END_IF

_sTemp := Tc2_Standard.MID(_sString, _nLength, nPosition);
IF (_nOffset := Tc2_Standard.FIND(_sTemp, sToFind)) <> 0 THEN
	nStart := nPosition + _nOffset - 1;
	nEnd := nPosition + _nOffset - 2 + Tc2_Standard.LEN(sToFind);
END_IF
END_METHOD

// Finds the last occurrence of a substring before the specified position.
// Outputs the start and end positions of the found substring.
METHOD FindLastBefore : I_Strb
VAR_INPUT
    sToFind : Str;        // Substring to find
    nPosition : INT := 256; // Starting position for reverse search
END_VAR
VAR_OUTPUT
    nStart : INT;         // Start position of the found substring
    nEnd : INT;           // End position of the found substring
END_VAR
VAR
	_sTemp			: Str;
	_nFindLength	: INT := Tc2_Standard.LEN(sToFind);
	_nOffset		: INT;
END_VAR
FindLastBefore := _this;

IF sToFind = '' THEN
	RETURN;
END_IF

IF nPosition = 0 THEN
	RETURN;
END_IF

IF nPosition = 256 THEN
	nPosition := _nLength;
END_IF

REPEAT
	_sTemp := Tc2_Standard.MID(_sString, _nFindLength, nPosition);
	IF _sTemp = sToFind THEN
		nStart 	:= nPosition;
		nEnd	:= nPosition + _nFindLength - 1;
		RETURN;
	END_IF
UNTIL
	(nPosition := nPosition - 1) <= 0
END_REPEAT
END_METHOD

// Checks if the specified substring exists after the given position.
METHOD HasAfter : BOOL
VAR_INPUT
    sToFind : Str;      // Substring to search for
    nPosition : INT := 0; // Starting position for search
END_VAR
VAR_OUTPUT
    nStart : INT;       // Start position of the found substring
    nEnd : INT;         // End position of the found substring
END_VAR
FindFirstAfter(sToFind, nPosition, nStart => nStart, nEnd => nEnd);
HasAfter := nStart > 0;
END_METHOD

// Checks if the specified substring exists before the given position.
METHOD HasBefore : BOOL
VAR_INPUT
    sToFind : Str;        // Substring to search for
    nPosition : INT := 256; // Ending position for reverse search
END_VAR
VAR_OUTPUT
    nStart : INT;         // Start position of the found substring
    nEnd : INT;           // End position of the found substring
END_VAR
IF nPosition = 256 THEN
	nPosition := Tc2_Standard.LEN(_sString);
END_IF

FindLastBefore(sToFind, nPosition, nStart => nStart, nEnd => nEnd);
HasBefore := nStart > 0;
END_METHOD

// Inserts a specified substring at a given position.
// Truncates if the total length exceeds 255 characters.
METHOD Inject : I_Strb
VAR_INPUT
    nPosition : INT;    // Position to inject the string
    sToInject : Str;    // String to inject
END_VAR
VAR
	_nNewLength	: INT;
END_VAR
Inject := _this;

IF sToInject = '' THEN
	RETURN;
END_IF

IF nPosition = 0 THEN
	RETURN;
END_IF

IF nPosition > _nLength THEN
	RETURN;
END_IF

_nNewLength := Tc2_Standard.LEN(sToInject) + _nLength;
IF _nNewLength > 255 THEN
	_nNewLength := 255;
END_IF

_sString := Tc2_Standard.INSERT(_sString, sToInject, nPosition);
_nLength := _nNewLength;
END_METHOD

// Checks if the current string is empty.
METHOD IsEmpty : BOOL
VAR_INPUT
END_VAR
IsEmpty := _nLength = 0;
END_METHOD

// Returns the current length of the string.
// The length of the string is stored as a separate variable (_nLength) 
// and reflects the actual length of the content.
// Unlike Tc2_Standard.LEN(), which counts up to the first null character, 
// this method directly returns the stored length.
METHOD Length : INT
VAR_INPUT
END_VAR
Length := _nLength;
END_METHOD

// Prepends the specified string to the current string.
// Truncates if the total length exceeds 255 characters.
METHOD Prepend : I_Strb
VAR_INPUT
    sToAdd : Str; // String to prepend
END_VAR
VAR
	_nNewLength	: INT;
END_VAR
Prepend := _this;

IF sToAdd = '' THEN
	RETURN;
END_IF

_nNewLength := Tc2_Standard.LEN(sToAdd) + _nLength;
IF _nNewLength > 255 THEN
	_nNewLength := 255;
END_IF

_sString := Tc2_Standard.CONCAT(sToAdd, _sString);
_nLength := _nNewLength;
END_METHOD

// Returns the current string value.
METHOD Read : Str
VAR_INPUT
END_VAR
Read := _sString;
END_METHOD

// Removes a substring of specified length starting at a given position.
METHOD Remove : I_Strb
VAR_INPUT
    nLength : INT;    // Length of the substring to remove
    nPosition : INT;  // Starting position of the substring to remove
END_VAR

VAR
	_nPosition	: INT;
END_VAR
Remove := _this;

IF nPosition = 0 THEN
	RETURN;
END_IF

IF nPosition > _nLength THEN
	RETURN;
END_IF

IF nLength = 0 THEN
	RETURN;
END_IF

IF nLength + nPosition > _nLength THEN
	nLength := _nLength - nPosition + 1;
END_IF

_sString := Tc2_Standard.DELETE(_sString, nLength, nPosition);
_nLength := _nLength - nLength;
END_METHOD

// Sets the current string to a new value.
METHOD Set : I_Strb
VAR_INPUT
    sLiteral : Str; // New string value
END_VAR
Set 		:= _this;

_sString 	:= sLiteral;
_nLength	:= Tc2_Standard.LEN(sLiteral);
END_METHOD

// Extracts a substring starting from a given position with a specified length.
METHOD Slice : I_Strb
VAR_INPUT
    nLength : INT;   // Length of the slice
    nPosition : INT; // Starting position of the slice
END_VAR
VAR_OUTPUT
    sSlice : Strb;   // The sliced string
END_VAR
Slice := _this;

IF nPosition = 0 THEN
	RETURN;
END_IF

IF nLength = 0 THEN
	RETURN;
END_IF

sSlice.Set(Tc2_Standard.MID(_sString, nLength, nPosition));
END_METHOD

// Splits the string into two parts at the specified position.
METHOD Split : I_Strb
VAR_INPUT
    nPosition : INT; // Position to split the string
END_VAR
VAR_OUTPUT
    sLeft : Strb;    // Left part of the split
    sRight : Strb;   // Right part of the split
END_VAR
Split := _this;

IF nPosition = 0 THEN
	RETURN;
END_IF

sLeft.Set(Tc2_Standard.LEFT(_sString, nPosition));
sRight.Set(Tc2_Standard.RIGHT(_sString, _nLength - nPosition));
END_METHOD

END_FUNCTION_BLOCK

// ---- Strings/Strf/Strf.TcPOU
// The Strf provides utilities for string formatting.
PROGRAM Strf

// Formats a string using Tc2_Utilities.FB_FormatString with a single argument.
METHOD Fmt : Str
VAR_INPUT
	sFormat			: Str; // Format, check format specification on Beckhoff infosys.
	tcArg			: Tc2_Utilities.T_Arg;
END_VAR
VAR
	_fmt			: Tc2_Utilities.FB_FormatString;
END_VAR
_fmt(sFormat := sFormat, arg1 := tcArg, sOut => Fmt);
END_METHOD

// Adds left and/or right padding to a string with a specified fill character.
// Returns the padded string.
METHOD Padding : Str
VAR_INPUT
    sValue       : Str;  // The original string
    nLeftPadding : USINT := 0; // Number of padding characters to add to the left
    nRightPadding: USINT := 0; // Number of padding characters to add to the right
    sFillChar    : Ch := ' ';  // Character used for padding
END_VAR
VAR
	_nLen		: INT := Tc2_Standard.LEN(sValue);
	_nLeftMiss	: INT;
	_nRightMiss	: INT;	

	i			: INT;
END_VAR
_nLeftMiss := nLeftPadding - _nLen;
_nRightMiss := nRightPadding - _nLen;

IF _nLeftMiss > 0 THEN
	FOR i := 1 TO _nleftMiss DO
		sValue := Tc2_Standard.CONCAT(sFillChar, sValue);
	END_FOR	
END_IF

IF _nRightMiss > 0 THEN
	FOR i := 1 TO _nRightMiss DO
		sValue := Tc2_Standard.CONCAT(sFillChar, sValue);
	END_FOR	
END_IF

Padding := sValue;
END_METHOD

// Converts a TIME value to a human-readable string with specified minimum and maximum units.
// Returns the formatted time string.
METHOD SimpleTime : Str
VAR_INPUT
    tValue   : TIME;  // Time value to convert
    sMinUnit : Str := 'MS'; // Minimum unit (e.g., MS, S, M, H, D)
    sMaxUnit : Str := 'S';  // Maximum unit (e.g., MS, S, M, H, D)
END_VAR
VAR
	_nMinUnit	: USINT;
	_nMaxUnit	: USINT;
	_sValues	: ARRAY[1..5] OF Strb;
	_nValues	: ARRAY[1..5] OF UINT;
	_sUnits   	: ARRAY[1..5] OF STRING := ['MS', 'S', 'M', 'H', 'D'];
	_stTime		: Tc2_Utilities.OTSTRUCT;
	_i			: USINT;
	_strb		: Strb;
END_VAR
FOR _i := 1 TO 5 DO
	IF _sUnits[_i] = sMinUnit THEN
		_nMinUnit := _i;
	END_IF
	IF _sUnits[_i] = sMaxUnit THEN
		_nMaxUnit := _i;
	END_IF
END_FOR

IF _nMaxUnit = 0 THEN
	RETURN;
END_IF

IF _nMinUnit = 0 THEN
	RETURN;
END_IF

IF _nMinUnit > _nMaxUnit THEN
	RETURN;
END_IF

_stTime := Tc2_Utilities.TIME_TO_OTSTRUCT(tValue);
_stTime.wDay := _stTime.wWeek * 7 + _stTime.wDay;

_nValues[1] := WORD_TO_UINT(_stTime.wMilliseconds);
_nValues[2] := WORD_TO_UINT(_stTime.wSecond);
_nValues[3] := WORD_TO_UINT(_stTime.wMinute);
_nValues[4] := WORD_TO_UINT(_stTime.wHour);
_nValues[5] := WORD_TO_UINT(_stTime.wDay);

_sValues[1].Set(Strf.Padding(UINT_TO_STRING(_nValues[1]), 3, 0, '0')).Append('ms');
_sValues[2].Set(Strf.Padding(UINT_TO_STRING(_nValues[2]), 2, 0, '0')).Append('s');
_sValues[3].Set(Strf.Padding(UINT_TO_STRING(_nValues[3]), 2, 0, '0')).Append('m');
_sValues[4].Set(Strf.Padding(UINT_TO_STRING(_nValues[4]), 2, 0, '0')).Append('h');
_sValues[5].Set(Strf.Padding(UINT_TO_STRING(_nValues[5]), 3, 0, '0')).Append('d');

IF _nMaxUnit < 5 THEN
    FOR _i := 5 TO _nMaxUnit + 1 BY -1 DO
        IF _nValues[_i] <> 0 THEN
            _strb.Append(_sValues[_i].Read()).Append(' ');
        END_IF
    END_FOR
END_IF

FOR _i := _nMaxUnit TO _nMinUnit BY -1 DO
    _strb.Append(_sValues[_i].Read()).Append(' ');
END_FOR

SimpleTime := _strb.Read();
END_METHOD

END_PROGRAM

// ---- Tags/Casts/IArgToITag.TcPOU
(*
Casts I_Arg as I_Tag.
Returns:
- Ok - Success,
- Err.InvRef - Invalid reference,
- Err.Itf0 - Invalid interface,
- Err.NoMatch - Cast failed
*)
FUNCTION IArgToITag : Result
VAR_INPUT
	iIn		: I_Arg;
	iOut	: REFERENCE TO I_Tag;
END_VAR

IF NOT __ISVALIDREF(iOut) THEN
	IArgToITag := Err.InvRef;
	RETURN;
END_IF

IF iIn = 0 THEN
	IArgToITag := Err.Itf0;
	RETURN;
END_IF

IF __QUERYINTERFACE(iIn, iOut) THEN
	IArgToITag := Ok;
ELSE
	IArgToITag := Err.NoMatch;
END_IF

END_FUNCTION

// ---- Tags/Helpers/GetTag.TcPOU
(*
Searches an `I_Entity` for a `I_Tag` component matching provided id pattern.
Result:
- Ok - Returns iTag.
- Err.NotFound - Returns null.
- Err.InvRef - Provided reference is invalid.
- Err.Itf0 - Returns null, incorrect interface.
*)
FUNCTION GetTag : Result
VAR_INPUT
	iEntity		: I_Entity;
	sIdPattern	: Str;
	iOut		: REFERENCE TO I_Tag;
END_VAR
VAR
	_iComp		: I_Component;
	cmp			: TagCmp;
END_VAR

IF iEntity = 0 THEN
	GetTag := Err.Itf0;
	RETURN;
END_IF

IF NOT __ISVALIDREF(iOut) THEN
	GetTag := Err.InvRef;
	RETURN;
END_IF

WHILE IsOk(iEntity.GetNextComp(_iComp)) DO
	IF IsOk(ICompToITag(_iComp.Raw, iOut)) THEN
		IF cmp.Set(iOut).MatchWcdId(sIdPattern).IsTrue() THEN
			GetTag := Ok;
			RETURN;
		ELSE
			iOut := 0;
		END_IF
	END_IF
END_WHILE

GetTag := Err.NotFound;

END_FUNCTION

// ---- Tags/Helpers/GetTagOption.TcPOU
(*
Searches an `I_Entity` for a `I_Tag` component with provided `Option` value.
Result:
- Ok - Returns iTag.
- Err.NotFound - Returns null.
- Err.InvRef - Provided reference is invalid.
- Err.Itf0 - Returns null, incorrect interface.
*)
FUNCTION GetTagOption : Result
VAR_INPUT
	iEntity		: I_Entity;
	sOption		: Str;
	iOut		: REFERENCE TO I_Tag;
END_VAR
VAR
	_iComp		: I_Component;
END_VAR

IF iEntity = 0 THEN
	GetTagOption := Err.Itf0;
	RETURN;
END_IF

IF NOT __ISVALIDREF(iOut) THEN
	GetTagOption := Err.InvRef;
	RETURN;
END_IF

WHILE IsOk(iEntity.GetNextComp(_iComp)) DO
	IF IsOk(ICompToITag(_iComp.Raw, iOut)) THEN
		IF iOut.Option = sOption THEN
			GetTagOption := Ok;
			RETURN;
		ELSE
			iOut := 0;
		END_IF
	END_IF
END_WHILE

GetTagOption := Err.NotFound;

END_FUNCTION

// ---- Tags/Helpers/HasTagOption.TcPOU
(*
Searches an `I_Entity` for a `I_Tag` component with provided `Option` value.
Result:
- Ok
- Err.NotFound - Returns null.
- Err.Itf0 - Returns null, incorrect interface.
*)
FUNCTION HasTagOption : Result
VAR_INPUT
	iEntity		: I_Entity;
	sOption		: Str;
END_VAR
VAR
	_iComp		: I_Component;
	_iTag		: I_Tag;
END_VAR

IF iEntity = 0 THEN
	HasTagOption := Err.Itf0;
	RETURN;
END_IF

WHILE IsOk(iEntity.GetNextComp(_iComp)) DO
	IF IsOk(ICompToITag(_iComp.Raw, _iTag)) THEN
		IF _iTag.Option = sOption THEN
			HasTagOption := Ok;
			RETURN;
		END_IF
	END_IF
END_WHILE

HasTagOption := Err.NotFound;

END_FUNCTION

// ---- Tags/Helpers/MatchPath.TcPOU
(*
Returns whether the symbol's path matches the provided pattern.
Allows wildcards in form of "*" that can cover multiple segments.
Example pattern: *.functionBlock.*.bBool
Returns 'Ok' or 'Err.NoMatch'
*)
FUNCTION MatchPath : Result
VAR_INPUT
    sAddress : Str;  /// The symbol's path to evaluate
    sPattern : Str;  /// The pattern to match against
END_VAR
VAR
	pttPath				: TagPath;
	pttSeg				: Str;
	pttPeek				: Str;
	addPath				: TagPath;
	addSeg				: Str;
	bMatch				: BOOL;
END_VAR

// Init
IF IsErr(addPath.Set(sAddress)) THEN
	MatchPath := Err.NoMatch;
	RETURN;
END_IF
IF IsErr(pttPath.Set(sPattern)) THEN
	MatchPath := Err.NoMatch;
	RETURN;
END_IF

// Advance to the next segment
WHILE IsOk(pttPath.Next(sSeg => pttSeg)) DO	
	bMatch := FALSE;
	// If the current segment is a wildcard, then peek to the next segment
	IF pttSeg = '*' THEN
		IF IsOk(pttPath.Peek(sSeg => pttPeek)) THEN
			IF pttPeek = '*' THEN
				CONTINUE; // Skip redundant wildcard if *.*.
			END_IF
		ELSE
			MatchPath := Ok;
			RETURN; // No more segments in the pattern, so it's a match as everything so far matched(.*)
		END_IF

	// If current segment is not a wildcard reset the peek.
	ELSIF pttSeg <> '*' THEN
		pttPeek := '';
	END_IF
	
	// Get the next segment of the address path
	WHILE IsOk(addPath.Next(sSeg => addSeg)) DO
		IF pttPeek <> '' THEN
			IF pttPeek = addSeg THEN
				bMatch := TRUE;
				pttPath.Next(); // Consume get next pattern segment
				EXIT;
			ELSE
				CONTINUE; // Get next address
			END_IF
		ELSIF pttSeg = addSeg THEN
			bMatch := TRUE;
			EXIT; // Consume get next pattern segment
		ELSE
			MatchPath := Err.NoMatch;
			RETURN; // No match - return
		END_IF
	END_WHILE

	IF NOT bMatch THEN
		MatchPath := Err.NoMatch;
		RETURN;
	END_IF

END_WHILE

IF IsOk(addPath.Peek()) THEN
	MatchPath := Err.NoMatch;
	RETURN;
END_IF

MatchPath := Ok;

END_FUNCTION

// ---- Jobs/Worker/Base/Worker.TcPOU
(*
Schedules jobs execution.
*)
FUNCTION_BLOCK Worker IMPLEMENTS I_Worker
VAR
	_iFirst: I_Job;
	_iLast: I_Job;	
END_VAR

(*
Defer the Job. Move it to the end of queue.
Returns:
- Ok - Success
- Err.Itf0 - iJob = 0
- Err.NoMatch = iJob.Worker <> THIS^
*)
METHOD Defer : Result
VAR_INPUT
    iJob : I_Job;
END_VAR
VAR
    _iPrev  : I_Job;
    _iNext  : I_Job;
    _iThis  : I_Worker := THIS^;
END_VAR
IF iJob = 0 THEN
    Defer := Err.Itf0;
    RETURN;
END_IF;

IF iJob.Worker <> _iThis THEN
    Defer := Err.NoMatch;
    RETURN;
END_IF;

_iPrev := iJob._Prev;
_iNext := iJob._Next;

IF _iPrev <> 0 THEN
    _iPrev._Next := _iNext;
ELSE
    _iFirst := _iNext;
END_IF;

IF _iNext <> 0 THEN
    _iNext._Prev := _iPrev;
ELSE
    _iLast := _iPrev;
END_IF;

iJob._Prev := _iLast;
iJob._Next := 0;

IF _iLast <> 0 THEN
    _iLast._Next := iJob;
ELSE
    _iFirst := iJob;
END_IF;

_iLast := iJob;

Defer := Ok;
END_METHOD

(*
Remove job from the queue and resets it.
Returns:
- Ok - Success
- Err.Itf0 - iJob = 0
- Err.NoMatch - iJob.Worker <> THIS^
- Err.IncArg - iJob.State = TaskState.Idle
*)
METHOD Dequeue : Result
VAR_INPUT
	iJob: I_Job;
END_VAR
VAR
	_iPrev: I_Job;
	_iNext: I_Job;
	_iThis: I_Worker := THIS^;
END_VAR
IF iJob = 0 THEN
	Dequeue := Err.Itf0;
    RETURN;
END_IF;

IF iJob.Worker <> _iThis THEN
    Dequeue := Err.NoMatch;
    RETURN;
END_IF;

IF iJob.State = JobState.Idle THEN
    Dequeue := Err.IncArg;
    RETURN;
END_IF;

_iPrev := iJob._Prev;
_iNext := iJob._Next;

IF _iPrev <> 0 THEN
    _iPrev._Next := _iNext;
ELSE
    _iFirst := _iNext;
END_IF;

IF _iNext <> 0 THEN
    _iNext._Prev := _iPrev;
ELSE
    _iLast := _iPrev;
END_IF;

IF iJob.State = JobState.Completed THEN
	iJob._OnDone();
ELSIF iJob.State = JobState.Aborted THEN
	iJob._OnAbort();
END_IF

iJob._OnExit();
Dequeue := Ok;
END_METHOD

(*
Add Job to queue.
Returns:
- Ok - Success
- Err.Itf0 - iJob = 0
- Err.NoMatch - iJob.Worker <> THIS^
- Err.IncArg - iJob.State <> TaskState.Idle 
*)
METHOD Enqueue : Result
VAR_INPUT
	iJob: I_Job;
END_VAR
VAR
	_iThis: I_Worker := THIS^;
END_VAR
IF iJob = 0 THEN
    Enqueue := Err.Itf0;
    RETURN;
END_IF;

IF iJob.Worker <> _iThis THEN
    Enqueue := Err.NoMatch;
    RETURN;
END_IF;

IF iJob.State <> JobState.Idle THEN
    Enqueue := Err.IncArg;
    RETURN;
END_IF;

iJob._Prev := _iLast;
iJob._Next := 0;
IF _iLast <> 0 THEN
    _iLast._Next := iJob;
ELSE
    _iFirst := iJob;
END_IF;
_iLast := iJob;

iJob._OnStart();
Enqueue := Ok;
END_METHOD

(*
Returns first the Job in queue.
*)
PROPERTY First : I_Job
GET
First := _iFirst;
END_GET
END_PROPERTY

(*
Runs Worker.
*)
METHOD Run : Result
VAR_INPUT
	iJob	: I_Job;
END_VAR
IF iJob <> 0 THEN
	CASE iJob.State OF
		JobState.Aborted:
			Run := Ok;
		
		JobState.Completed:
			Run := Ok;	
		
		JobState.Ready:
			iJob._OnRun();
			Run := Ok;
	
		JobState.Error, JobState.Idle, JobState.Running:
			Run := Err.IncArg;
			
	END_CASE
ELSE
	Run := Err.Itf0;
END_IF
END_METHOD

END_FUNCTION_BLOCK

// ---- Jobs/Worker/LoopWorker.TcPOU
(*
Worker wrapper that runs different job each on iteration.
*)
FUNCTION_BLOCK LoopWorker
VAR
	_scheduler: Worker;
END_VAR

(*
Returns internal Worker.
*)
PROPERTY Base : I_Worker
GET
Base := _scheduler;
END_GET
END_PROPERTY

METHOD Run
VAR_INPUT
END_VAR
IF _scheduler.First = 0 THEN
	RETURN;
END_IF

CASE _scheduler.First.State OF
	JobState.Completed, JobState.Aborted:
		_scheduler.Dequeue(_scheduler.First);
END_CASE

CASE _scheduler.Run(_scheduler.First) OF
	Ok:
		_scheduler.Defer(_scheduler.First);
	Err.Itf0:
		RETURN;
	ELSE
		NewDebug(_scheduler, Param.EXE_INTERNAL_DEBUG_MODE, 'Scheduler: Incorrect task state!', _scheduler.First);
		RETURN;	
END_CASE
END_METHOD

END_FUNCTION_BLOCK

// ---- Jobs/Worker/BlockingWorker.TcPOU
(*
Worker wrapper that runs job until completition.
*)
FUNCTION_BLOCK BlockingWorker
VAR
	_scheduler: Worker;
END_VAR

(*
Returns internal Worker.
*)
PROPERTY Base : I_Worker
GET
Base := _scheduler;
END_GET
END_PROPERTY

METHOD Run
VAR_INPUT
END_VAR
IF _scheduler.First = 0 THEN
	RETURN;
END_IF

CASE _scheduler.First.State OF
	JobState.Completed, JobState.Aborted:
		_scheduler.Dequeue(_scheduler.First);
END_CASE

CASE _scheduler.Run(_scheduler.First) OF
	Ok:
		// Do Nothing
	Err.Itf0:
		RETURN;
	ELSE
		NewDebug(_scheduler, Param.EXE_INTERNAL_DEBUG_MODE, 'Scheduler: Incorrect task state!', _scheduler.First);
		RETURN;	
END_CASE
END_METHOD

END_FUNCTION_BLOCK

// ---- Jobs/Job/Job.TcPOU
(*
An abstract representation of a system job, providing the foundation for implementing job-specific behavior. Manages its state.  
Offers default behavior for its lifecycle methods, allowing programmers to override only the relevant parts.
*)
FUNCTION_BLOCK ABSTRACT Job IMPLEMENTS I_Job
VAR
	{attribute 'hide'}
	_iNext: I_Job;
	{attribute 'hide'}
	_iPrev: I_Job;
	{attribute 'hide'}
	_iWorker: I_Worker;
	{attribute 'hide'}
	_eState: JobState;
	
	
END_VAR

PROPERTY INTERNAL _Next : I_Job
GET
_Next := _iNext;
END_GET
SET
_iNext := _Next;
END_SET
END_PROPERTY

METHOD INTERNAL _OnAbort
VAR_INPUT
END_VAR
OnAbort();
END_METHOD

METHOD INTERNAL _OnDone
VAR_INPUT
END_VAR
OnDone();
END_METHOD

METHOD INTERNAL _OnExit
VAR_INPUT
END_VAR
_iNext := 0;
_iPrev := 0;
_eState := JobState.Idle;
OnExit();
END_METHOD

METHOD INTERNAL _OnRun
VAR_INPUT
END_VAR
_eState := JobState.Running;
OnRun();
IF _eState = JobState.Running THEN
	_eState := JobState.Ready;
END_IF
END_METHOD

METHOD INTERNAL _OnStart
VAR_INPUT
END_VAR
OnStart();
END_METHOD

PROPERTY INTERNAL _Prev : I_Job
GET
_Prev := _iPrev;
END_GET
SET
_iPrev := _Prev;
END_SET
END_PROPERTY

(*
Notifies scheduler to aboort this job.
Returns Err.IncArg on State = Idle
*)
METHOD Abort : Result
VAR_INPUT
END_VAR
IF _eState = JobState.Idle THEN
	Abort := Err.IncArg;
	RETURN;
END_IF

_eState := JobState.Aborted;
Abort := Ok;
END_METHOD

(*
Notifies scheduler that the jobs is completed.
Returns Err.IncArg on State <> Running
*)
METHOD PROTECTED Done : Result
VAR_INPUT
END_VAR
IF _eState <> JobState.Running THEN
	Done := Err.IncArg;
	RETURN;
END_IF

_eState := JobState.Completed;
Done := Ok;
END_METHOD

(*
Executed when this job is aborted.  
*)
METHOD PROTECTED OnAbort
VAR_INPUT
END_VAR
END_METHOD

(*
Executed when this job is done.  
*)
METHOD PROTECTED OnDone
VAR_INPUT
END_VAR
END_METHOD

(*
Executed when this job is dequeued.  
*)
METHOD PROTECTED OnExit
VAR_INPUT
END_VAR
END_METHOD

(*
Executed when this job is run.  
*)
METHOD PROTECTED OnRun
VAR_INPUT
END_VAR
END_METHOD

(*
Executed when this job is started.  
*)
METHOD PROTECTED OnStart
VAR_INPUT
END_VAR
END_METHOD

(*
Starts the job and adds it to Workers queue.
Returns Err.IncArg on State <> Idle.
Returns Err.Itf0 on Worker = 0.
*)
METHOD Start : Result
VAR_INPUT
END_VAR
IF _eState <> JobState.Idle THEN
	Start := Err.IncArg;
	RETURN;
END_IF

IF _iWorker = 0 THEN
	Start := Err.Itf0;
	RETURN;
END_IF

IF IsOk(_iWorker.Enqueue(THIS^), nOut => Start) THEN
	_eState := JobState.Ready;
END_IF
END_METHOD

(*
Returns Jobs state
*)
PROPERTY State : JobState
GET
State := _eState;
END_GET
END_PROPERTY

(*
Returns Worker working on this job
*)
PROPERTY Worker : I_Worker
GET
Worker := _iWorker;
END_GET
SET
IF _eState = JobState.Idle THEN
	_iWorker := Worker;
END_IF
END_SET
END_PROPERTY

END_FUNCTION_BLOCK
